LIN {X 0,Y 318.098,Z 206.968,A -85,B 0,C 180,E1 -15903.08,E2 -15903.08} C_VEL
LIN {X 0,Y 320.749,Z 222.526,A -85,B 0,C 180,E1 -15903.782,E2 -15903.782} C_VEL
LIN {X 0,Y 321.576,Z 229.62,A -85,B 0,C 180,E1 -15904.057,E2 -15904.057} C_VEL
LIN {X 0,Y 319.669,Z 290.634,A -85,B 0,C 180,E1 -15905.482,E2 -15905.482} C_VEL
LIN {X 0,Y 318.704,Z 303.737,A -85,B 0,C 180,E1 -15906.01,E2 -15906.01} C_VEL
LIN {X 0,Y 317.246,Z 316.408,A -85,B 0,C 180,E1 -15906.759,E2 -15906.759} C_VEL
LIN {X 0,Y 315.532,Z 328.526,A -85,B 0,C 180,E1 -15907.75,E2 -15907.75} C_VEL
LIN {X 0,Y 313.654,Z 340.033,A -85,B 0,C 180,E1 -15908.991,E2 -15908.991} C_VEL
LIN {X 0,Y 311.666,Z 350.433,A -85,B 0,C 180,E1 -15910.401,E2 -15910.401} C_VEL
LIN {X 0,Y 309.931,Z 358.976,A -85,B 0,C 180,E1 -15911.832,E2 -15911.832} C_VEL
LIN {X 0,Y 308.237,Z 367.598,A -85,B 0,C 180,E1 -15913.609,E2 -15913.609} C_VEL
LIN {X 0,Y 306.912,Z 374.656,A -85,B 0,C 180,E1 -15915.41,E2 -15915.41} C_VEL
LIN {X 0,Y 305.513,Z 380.916,A -85,B 0,C 180,E1 -15917.377,E2 -15917.377} C_VEL
LIN {X 0,Y 304.63,Z 385.925,A -85,B 0,C 180,E1 -15919.364,E2 -15919.364} C_VEL
LIN {X 0,Y 304.053,Z 389.825,A -85,B 0,C 180,E1 -15921.359,E2 -15921.359} C_VEL
LIN {X 0,Y 303.728,Z 392.717,A -85,B 0,C 180,E1 -15923.356,E2 -15923.356} C_VEL
LIN {X 0,Y 303.654,Z 395.096,A -85,B 0,C 180,E1 -15926.018,E2 -15926.018} C_VEL
LIN {X 0,Y 303.656,Z 395.702,A -85,B 0,C 180,E1 -15927.347,E2 -15927.347} C_VEL
LIN {X 0,Y 303.684,Z 395.883,A -85,B 0,C 180,E1 -15928.674,E2 -15928.674} C_VEL
LIN {X 0,Y 303.769,Z 395.655,A -85,B 0,C 180,E1 -15930,E2 -15930} C_VEL
LIN {X 0,Y 303.713,Z 395.029,A -85,B 0,C 180,E1 -15931.326,E2 -15931.326} C_VEL
LIN {X 0,Y 303.684,Z 394.007,A -85,B 0,C 180,E1 -15932.653,E2 -15932.653} C_VEL
LIN {X 0,Y 303.693,Z 392.539,A -85,B 0,C 180,E1 -15933.981,E2 -15933.981} C_VEL
LIN {X 0,Y 303.678,Z 390.075,A -85,B 0,C 180,E1 -15935.644,E2 -15935.644} C_VEL
LIN {X 0,Y 303.905,Z 385.397,A -85,B 0,C 180,E1 -15937.975,E2 -15937.975} C_VEL
LIN {X 0,Y 304.352,Z 379.061,A -85,B 0,C 180,E1 -15940.309,E2 -15940.309} C_VEL
LIN {X 0,Y 305.069,Z 372.151,A -85,B 0,C 180,E1 -15942.304,E2 -15942.304} C_VEL
LIN {X 0,Y 305.868,Z 365.084,A -85,B 0,C 180,E1 -15943.961,E2 -15943.961} C_VEL
LIN {X 0,Y 306.783,Z 357.329,A -85,B 0,C 180,E1 -15945.47,E2 -15945.47} C_VEL
LIN {X 0,Y 307.987,Z 347.315,A -85,B 0,C 180,E1 -15947.068,E2 -15947.068} C_VEL
LIN {X 0,Y 309.154,Z 336.997,A -85,B 0,C 180,E1 -15948.386,E2 -15948.386} C_VEL
LIN {X 0,Y 310.341,Z 325.889,A -85,B 0,C 180,E1 -15949.513,E2 -15949.513} C_VEL
LIN {X 0,Y 311.511,Z 313.595,A -85,B 0,C 180,E1 -15950.468,E2 -15950.468} C_VEL
LIN {X 0,Y 312.47,Z 300.68,A -85,B 0,C 180,E1 -15951.178,E2 -15951.178} C_VEL
LIN {X 0,Y 313.032,Z 286.986,A -85,B 0,C 180,E1 -15951.656,E2 -15951.656} C_VEL
LIN {X 0,Y 314.192,Z 225.236,A -85,B 0,C 180,E1 -15953.088,E2 -15953.088} C_VEL
LIN {X 0,Y 308.653,Z 182.969,A -85,B 0,C 180,E1 -15954.491,E2 -15954.491} C_VEL
LIN {X 0,Y 309.452,Z 175.908,A -85,B 0,C 180,E1 -15956.287,E2 -15956.287} C_VEL
LIN {X 0,Y 308.009,Z 167.396,A -85,B 0,C 180,E1 -15958.631,E2 -15958.631} C_VEL
LIN {X 0,Y 305.479,Z 155.435,A -85,B 0,C 180,E1 -15962.094,E2 -15962.094} C_VEL
LIN {X 0,Y 305.5,Z 155.431,A -85,B 0,C 180,E1 -15966.373,E2 -15966.373} C_VEL
LIN {X 0,Y 305.459,Z 155.436,A -85,B 0,C 180,E1 -15970.107,E2 -15970.107} C_VEL
LIN {X 0,Y 305.426,Z 155.442,A -85,B 0,C 180,E1 -15973.655,E2 -15973.655} C_VEL
LIN {X 0,Y 305.455,Z 155.437,A -85,B 0,C 180,E1 -15977.414,E2 -15977.414} C_VEL
LIN {X 0,Y 305.476,Z 155.437,A -85,B 0,C 180,E1 -15981.597,E2 -15981.597} C_VEL
LIN {X 0,Y 305.462,Z 155.434,A -85,B 0,C 180,E1 -15984.886,E2 -15984.886} C_VEL
LIN {X 0,Y 305.452,Z 155.434,A -85,B 0,C 180,E1 -15988.355,E2 -15988.355} C_VEL
LIN {X 0,Y 305.521,Z 155.429,A -85,B 0,C 180,E1 -15991.114,E2 -15991.114} C_VEL
LIN {X 0,Y 305.572,Z 155.419,A -85,B 0,C 180,E1 -15994.088,E2 -15994.088} C_VEL
LIN {X 0,Y 305.475,Z 155.429,A -85,B 0,C 180,E1 -15998.401,E2 -15998.401} C_VEL
LIN {X 0,Y 305.542,Z 155.417,A -85,B 0,C 180,E1 -16001.214,E2 -16001.214} C_VEL
LIN {X 0,Y 305.626,Z 155.412,A -85,B 0,C 180,E1 -16005.348,E2 -16005.348} C_VEL
LIN {X 0,Y 305.624,Z 155.413,A -85,B 0,C 180,E1 -16009.399,E2 -16009.399} C_VEL
LIN {X 0,Y 305.748,Z 155.396,A -85,B 0,C 180,E1 -16012.072,E2 -16012.072} C_VEL
LIN {X 0,Y 305.674,Z 155.407,A -85,B 0,C 180,E1 -16014.723,E2 -16014.723} C_VEL
LIN {X 0,Y 305.955,Z 155.375,A -85,B 0,C 180,E1 -16018.683,E2 -16018.683} C_VEL
LIN {X 0,Y 305.955,Z 155.368,A -85,B 0,C 180,E1 -16021.316,E2 -16021.316} C_VEL
LIN {X 0,Y 305.685,Z 155.404,A -85,B 0,C 180,E1 -16025.276,E2 -16025.276} C_VEL
LIN {X 0,Y 305.796,Z 155.391,A -85,B 0,C 180,E1 -16027.926,E2 -16027.926} C_VEL
LIN {X 0,Y 305.603,Z 155.412,A -85,B 0,C 180,E1 -16031.945,E2 -16031.945} C_VEL
LIN {X 0,Y 305.637,Z 155.411,A -85,B 0,C 180,E1 -16035.035,E2 -16035.035} C_VEL
LIN {X 0,Y 305.579,Z 155.418,A -85,B 0,C 180,E1 -16038.783,E2 -16038.783} C_VEL
LIN {X 0,Y 305.485,Z 155.428,A -85,B 0,C 180,E1 -16043.039,E2 -16043.039} C_VEL
LIN {X 0,Y 305.546,Z 155.426,A -85,B 0,C 180,E1 -16046.227,E2 -16046.227} C_VEL
LIN {X 0,Y 305.487,Z 155.427,A -85,B 0,C 180,E1 -16049.047,E2 -16049.047} C_VEL
LIN {X 0,Y 305.442,Z 155.438,A -85,B 0,C 180,E1 -16051.952,E2 -16051.952} C_VEL
LIN {X 0,Y 305.461,Z 155.432,A -85,B 0,C 180,E1 -16055.113,E2 -16055.113} C_VEL
LIN {X 0,Y 305.44,Z 155.433,A -85,B 0,C 180,E1 -16058.527,E2 -16058.527} C_VEL
LIN {X 0,Y 305.454,Z 155.433,A -85,B 0,C 180,E1 -16062.586,E2 -16062.586} C_VEL
LIN {X 0,Y 305.424,Z 155.437,A -85,B 0,C 180,E1 -16066.345,E2 -16066.345} C_VEL
LIN {X 0,Y 305.457,Z 155.435,A -85,B 0,C 180,E1 -16069.892,E2 -16069.892} C_VEL
LIN {X 0,Y 305.48,Z 155.434,A -85,B 0,C 180,E1 -16073.632,E2 -16073.632} C_VEL
LIN {X 0,Y 305.464,Z 155.431,A -85,B 0,C 180,E1 -16076.483,E2 -16076.483} C_VEL
LIN {X 0,Y 305.495,Z 155.43,A -85,B 0,C 180,E1 -16080.95,E2 -16080.95} C_VEL
LIN {X 0,Y 305.571,Z 155.418,A -85,B 0,C 180,E1 -16084.088,E2 -16084.088} C_VEL
LIN {X 0,Y 305.475,Z 155.432,A -85,B 0,C 180,E1 -16088.401,E2 -16088.401} C_VEL
LIN {X 0,Y 305.542,Z 155.425,A -85,B 0,C 180,E1 -16091.215,E2 -16091.215} C_VEL
LIN {X 0,Y 305.626,Z 155.414,A -85,B 0,C 180,E1 -16095.348,E2 -16095.348} C_VEL
LIN {X 0,Y 305.624,Z 155.414,A -85,B 0,C 180,E1 -16099.399,E2 -16099.399} C_VEL
LIN {X 0,Y 305.748,Z 155.395,A -85,B 0,C 180,E1 -16102.073,E2 -16102.073} C_VEL
LIN {X 0,Y 305.674,Z 155.541,A -85,B 0,C 180,E1 -16104.889,E2 -16104.889} C_VEL
LIN {X 0,Y 306.008,Z 157.231,A -85,B 0,C 180,E1 -16105.424,E2 -16105.424} C_VEL
LIN {X 0,Y 313.1,Z 177.176,A -85,B 0,C 180,E1 -16106.405,E2 -16106.405} C_VEL
LIN {X 0,Y 314.55,Z 182.856,A -85,B 0,C 180,E1 -16106.637,E2 -16106.637} C_VEL
LIN {X 0,Y 315.065,Z 186.672,A -85,B 0,C 180,E1 -16106.763,E2 -16106.763} C_VEL
LIN {X 0,Y 313.152,Z 265.366,A -85,B 0,C 180,E1 -16108.599,E2 -16108.599} C_VEL
LIN {X 0,Y 312.585,Z 278.914,A -85,B 0,C 180,E1 -16109.195,E2 -16109.195} C_VEL
LIN {X 0,Y 311.853,Z 291.275,A -85,B 0,C 180,E1 -16110,E2 -16110} C_VEL
LIN {X 0,Y 310.932,Z 302.407,A -85,B 0,C 180,E1 -16110.972,E2 -16110.972} C_VEL
LIN {X 0,Y 309.759,Z 313.993,A -85,B 0,C 180,E1 -16112.269,E2 -16112.269} C_VEL
LIN {X 0,Y 308.583,Z 324.524,A -85,B 0,C 180,E1 -16113.755,E2 -16113.755} C_VEL
LIN {X 0,Y 307.513,Z 333.085,A -85,B 0,C 180,E1 -16115.245,E2 -16115.245} C_VEL
LIN {X 0,Y 306.334,Z 342.342,A -85,B 0,C 180,E1 -16117.249,E2 -16117.249} C_VEL
LIN {X 0,Y 305.428,Z 349.79,A -85,B 0,C 180,E1 -16119.269,E2 -16119.269} C_VEL
LIN {X 0,Y 304.727,Z 355.732,A -85,B 0,C 180,E1 -16121.306,E2 -16121.306} C_VEL
LIN {X 0,Y 304.265,Z 360.38,A -85,B 0,C 180,E1 -16123.355,E2 -16123.355} C_VEL
LIN {X 0,Y 303.862,Z 363.912,A -85,B 0,C 180,E1 -16125.426,E2 -16125.426} C_VEL
LIN {X 0,Y 303.599,Z 367.109,A -85,B 0,C 180,E1 -16128.359,E2 -16128.359} C_VEL
LIN {X 0,Y 303.554,Z 368.119,A -85,B 0,C 180,E1 -16130.322,E2 -16130.322} C_VEL
LIN {X 0,Y 303.691,Z 368.27,A -85,B 0,C 180,E1 -16132.23,E2 -16132.23} C_VEL
LIN {X 0,Y 304.02,Z 367.364,A -85,B 0,C 180,E1 -16134.589,E2 -16134.589} C_VEL
LIN {X 0,Y 304.337,Z 366.189,A -85,B 0,C 180,E1 -16136.025,E2 -16136.025} C_VEL
LIN {X 0,Y 305.026,Z 363.501,A -85,B 0,C 180,E1 -16138.186,E2 -16138.186} C_VEL
LIN {X 0,Y 305.938,Z 359.612,A -85,B 0,C 180,E1 -16140.357,E2 -16140.357} C_VEL
LIN {X 0,Y 307.175,Z 354.217,A -85,B 0,C 180,E1 -16142.593,E2 -16142.593} C_VEL
LIN {X 0,Y 308.695,Z 347.638,A -85,B 0,C 180,E1 -16144.693,E2 -16144.693} C_VEL
LIN {X 0,Y 310.26,Z 340.559,A -85,B 0,C 180,E1 -16146.485,E2 -16146.485} C_VEL
LIN {X 0,Y 312.107,Z 331.396,A -85,B 0,C 180,E1 -16148.354,E2 -16148.354} C_VEL
LIN {X 0,Y 313.882,Z 322.187,A -85,B 0,C 180,E1 -16149.861,E2 -16149.861} C_VEL
LIN {X 0,Y 315.728,Z 311.658,A -85,B 0,C 180,E1 -16151.245,E2 -16151.245} C_VEL
LIN {X 0,Y 317.434,Z 299.665,A -85,B 0,C 180,E1 -16152.476,E2 -16152.476} C_VEL
LIN {X 0,Y 318.779,Z 287.425,A -85,B 0,C 180,E1 -16153.438,E2 -16153.438} C_VEL
LIN {X 0,Y 319.871,Z 274.616,A -85,B 0,C 180,E1 -16154.151,E2 -16154.151} C_VEL
LIN {X 0,Y 320.505,Z 261.159,A -85,B 0,C 180,E1 -16154.635,E2 -16154.635} C_VEL
LIN {X 0,Y 322.56,Z 192.231,A -85,B 0,C 180,E1 -16156.232,E2 -16156.232} C_VEL
LIN {X 0,Y 316.448,Z 178.489,A -85,B 0,C 180,E1 -16157.287,E2 -16157.287} C_VEL
LIN {X 0,Y 316.128,Z 177.812,A -85,B 0,C 180,E1 -16157.343,E2 -16157.343} C_VEL
LIN {X 0,Y 314.073,Z 174.928,A -85,B 0,C 180,E1 -16157.664,E2 -16157.664} C_VEL
LIN {X 0,Y 309.469,Z 171.568,A -85,B 0,C 180,E1 -16158.319,E2 -16158.319} C_VEL
LIN {X 0,Y 304.78,Z 168.323,A -85,B 0,C 180,E1 -16159.01,E2 -16159.01} C_VEL
LIN {X 0,Y 302.586,Z 165.592,A -85,B 0,C 180,E1 -16159.38,E2 -16159.38} C_VEL
LIN {X 0,Y 299.095,Z 159.067,A -85,B 0,C 180,E1 -16160.076,E2 -16160.076} C_VEL
LIN {X 0,Y 298.387,Z 156.315,A -85,B 0,C 180,E1 -16161.212,E2 -16161.212} C_VEL
LIN {X 0,Y 298.404,Z 156.303,A -85,B 0,C 180,E1 -16163.928,E2 -16163.928} C_VEL
LIN {X 0,Y 298.393,Z 156.318,A -85,B 0,C 180,E1 -16167.2,E2 -16167.2} C_VEL
LIN {X 0,Y 298.365,Z 156.321,A -85,B 0,C 180,E1 -16170.638,E2 -16170.638} C_VEL
LIN {X 0,Y 298.413,Z 156.312,A -85,B 0,C 180,E1 -16174.918,E2 -16174.918} C_VEL
LIN {X 0,Y 298.389,Z 156.309,A -85,B 0,C 180,E1 -16177.862,E2 -16177.862} C_VEL
LIN {X 0,Y 298.451,Z 156.301,A -85,B 0,C 180,E1 -16180.751,E2 -16180.751} C_VEL
LIN {X 0,Y 298.511,Z 156.292,A -85,B 0,C 180,E1 -16184.991,E2 -16184.991} C_VEL
LIN {X 0,Y 298.578,Z 156.28,A -85,B 0,C 180,E1 -16189.146,E2 -16189.146} C_VEL
LIN {X 0,Y 298.7,Z 156.276,A -85,B 0,C 180,E1 -16191.885,E2 -16191.885} C_VEL
LIN {X 0,Y 298.626,Z 156.28,A -85,B 0,C 180,E1 -16194.599,E2 -16194.599} C_VEL
LIN {X 0,Y 298.903,Z 156.24,A -85,B 0,C 180,E1 -16198.653,E2 -16198.653} C_VEL
LIN {X 0,Y 298.904,Z 156.25,A -85,B 0,C 180,E1 -16201.348,E2 -16201.348} C_VEL
LIN {X 0,Y 298.736,Z 156.268,A -85,B 0,C 180,E1 -16206.756,E2 -16206.756} C_VEL
LIN {X 0,Y 298.627,Z 156.283,A -85,B 0,C 180,E1 -16209.482,E2 -16209.482} C_VEL
LIN {X 0,Y 298.547,Z 156.286,A -85,B 0,C 180,E1 -16213.616,E2 -16213.616} C_VEL
LIN {X 0,Y 298.489,Z 156.3,A -85,B 0,C 180,E1 -16216.412,E2 -16216.412} C_VEL
LIN {X 0,Y 298.489,Z 156.304,A -85,B 0,C 180,E1 -16219.641,E2 -16219.641} C_VEL
LIN {X 0,Y 298.425,Z 156.308,A -85,B 0,C 180,E1 -16223.601,E2 -16223.601} C_VEL
LIN {X 0,Y 298.41,Z 156.303,A -85,B 0,C 180,E1 -16226.582,E2 -16226.582} C_VEL
LIN {X 0,Y 298.396,Z 156.31,A -85,B 0,C 180,E1 -16229.644,E2 -16229.644} C_VEL
LIN {X 0,Y 298.395,Z 156.316,A -85,B 0,C 180,E1 -16232.801,E2 -16232.801} C_VEL
LIN {X 0,Y 298.43,Z 156.307,A -85,B 0,C 180,E1 -16236.803,E2 -16236.803} C_VEL
LIN {X 0,Y 298.376,Z 156.318,A -85,B 0,C 180,E1 -16239.492,E2 -16239.492} C_VEL
LIN {X 0,Y 298.373,Z 156.317,A -85,B 0,C 180,E1 -16243.098,E2 -16243.098} C_VEL
LIN {X 0,Y 298.405,Z 156.32,A -85,B 0,C 180,E1 -16246.921,E2 -16246.921} C_VEL
LIN {X 0,Y 298.406,Z 156.317,A -85,B 0,C 180,E1 -16251.006,E2 -16251.006} C_VEL
LIN {X 0,Y 298.454,Z 156.374,A -85,B 0,C 180,E1 -16252.141,E2 -16252.141} C_VEL
LIN {X 0,Y 301.266,Z 166.786,A -85,B 0,C 180,E1 -16255.952,E2 -16255.952} C_VEL
LIN {X 0,Y 303.943,Z 178.256,A -85,B 0,C 180,E1 -16259.807,E2 -16259.807} C_VEL
LIN {X 0,Y 304.513,Z 181.202,A -85,B 0,C 180,E1 -16260.744,E2 -16260.744} C_VEL
LIN {X 0,Y 308.356,Z 190.471,A -85,B 0,C 180,E1 -16261.494,E2 -16261.494} C_VEL
LIN {X 0,Y 311.822,Z 206.926,A -85,B 0,C 180,E1 -16262.365,E2 -16262.365} C_VEL
LIN {X 0,Y 314.608,Z 223.163,A -85,B 0,C 180,E1 -16263.126,E2 -16263.126} C_VEL
LIN {X 0,Y 315.47,Z 230.001,A -85,B 0,C 180,E1 -16263.407,E2 -16263.407} C_VEL
LIN {X 0,Y 313.534,Z 290.112,A -85,B 0,C 180,E1 -16264.837,E2 -16264.837} C_VEL
LIN {X 0,Y 312.525,Z 303.285,A -85,B 0,C 180,E1 -16265.372,E2 -16265.372} C_VEL
LIN {X 0,Y 311.087,Z 315.427,A -85,B 0,C 180,E1 -16266.094,E2 -16266.094} C_VEL
LIN {X 0,Y 309.534,Z 326.016,A -85,B 0,C 180,E1 -16266.942,E2 -16266.942} C_VEL
LIN {X 0,Y 308.04,Z 335.282,A -85,B 0,C 180,E1 -16267.886,E2 -16267.886} C_VEL
LIN {X 0,Y 305.94,Z 346.581,A -85,B 0,C 180,E1 -16269.317,E2 -16269.317} C_VEL
LIN {X 0,Y 303.98,Z 355.709,A -85,B 0,C 180,E1 -16270.764,E2 -16270.764} C_VEL
LIN {X 0,Y 301.99,Z 364.922,A -85,B 0,C 180,E1 -16272.587,E2 -16272.587} C_VEL
LIN {X 0,Y 300.528,Z 372.301,A -85,B 0,C 180,E1 -16274.399,E2 -16274.399} C_VEL
LIN {X 0,Y 299.005,Z 378.958,A -85,B 0,C 180,E1 -16276.405,E2 -16276.405} C_VEL
LIN {X 0,Y 297.881,Z 384.307,A -85,B 0,C 180,E1 -16278.431,E2 -16278.431} C_VEL
LIN {X 0,Y 297.197,Z 388.504,A -85,B 0,C 180,E1 -16280.472,E2 -16280.472} C_VEL
LIN {X 0,Y 296.867,Z 390.741,A -85,B 0,C 180,E1 -16281.834,E2 -16281.834} C_VEL
LIN {X 0,Y 296.553,Z 393.862,A -85,B 0,C 180,E1 -16284.56,E2 -16284.56} C_VEL
LIN {X 0,Y 296.568,Z 394.833,A -85,B 0,C 180,E1 -16285.923,E2 -16285.923} C_VEL
LIN {X 0,Y 296.579,Z 395.406,A -85,B 0,C 180,E1 -16287.283,E2 -16287.283} C_VEL
LIN {X 0,Y 296.597,Z 395.544,A -85,B 0,C 180,E1 -16288.642,E2 -16288.642} C_VEL
LIN {X 0,Y 296.677,Z 395.291,A -85,B 0,C 180,E1 -16290,E2 -16290} C_VEL
LIN {X 0,Y 296.625,Z 394.64,A -85,B 0,C 180,E1 -16291.357,E2 -16291.357} C_VEL
LIN {X 0,Y 296.607,Z 393.588,A -85,B 0,C 180,E1 -16292.716,E2 -16292.716} C_VEL
LIN {X 0,Y 296.606,Z 392.071,A -85,B 0,C 180,E1 -16294.076,E2 -16294.076} C_VEL
LIN {X 0,Y 296.613,Z 388.985,A -85,B 0,C 180,E1 -16296.12,E2 -16296.12} C_VEL
LIN {X 0,Y 296.843,Z 384.814,A -85,B 0,C 180,E1 -16298.167,E2 -16298.167} C_VEL
LIN {X 0,Y 297.33,Z 378.412,A -85,B 0,C 180,E1 -16300.555,E2 -16300.555} C_VEL
LIN {X 0,Y 298.114,Z 371.432,A -85,B 0,C 180,E1 -16302.595,E2 -16302.595} C_VEL
LIN {X 0,Y 299.16,Z 362.658,A -85,B 0,C 180,E1 -16304.628,E2 -16304.628} C_VEL
LIN {X 0,Y 300.164,Z 353.634,A -85,B 0,C 180,E1 -16306.318,E2 -16306.318} C_VEL
LIN {X 0,Y 301.441,Z 343.735,A -85,B 0,C 180,E1 -16307.818,E2 -16307.818} C_VEL
LIN {X 0,Y 302.705,Z 332.818,A -85,B 0,C 180,E1 -16309.144,E2 -16309.144} C_VEL
LIN {X 0,Y 303.992,Z 320.561,A -85,B 0,C 180,E1 -16310.291,E2 -16310.291} C_VEL
LIN {X 0,Y 305.12,Z 307.747,A -85,B 0,C 180,E1 -16311.182,E2 -16311.182} C_VEL
LIN {X 0,Y 305.952,Z 294.977,A -85,B 0,C 180,E1 -16311.785,E2 -16311.785} C_VEL
LIN {X 0,Y 306.484,Z 277.039,A -85,B 0,C 180,E1 -16312.276,E2 -16312.276} C_VEL
LIN {X 0,Y 307.417,Z 225.576,A -85,B 0,C 180,E1 -16313.496,E2 -16313.496} C_VEL
LIN {X 0,Y 301.792,Z 182.64,A -85,B 0,C 180,E1 -16314.964,E2 -16314.964} C_VEL
LIN {X 0,Y 302.448,Z 176.485,A -85,B 0,C 180,E1 -16316.571,E2 -16316.571} C_VEL
LIN {X 0,Y 300.628,Z 166.507,A -85,B 0,C 180,E1 -16319.402,E2 -16319.402} C_VEL
LIN {X 0,Y 298.437,Z 156.311,A -85,B 0,C 180,E1 -16322.464,E2 -16322.464} C_VEL
LIN {X 0,Y 298.452,Z 156.308,A -85,B 0,C 180,E1 -16326.808,E2 -16326.808} C_VEL
LIN {X 0,Y 298.41,Z 156.314,A -85,B 0,C 180,E1 -16329.486,E2 -16329.486} C_VEL
LIN {X 0,Y 298.399,Z 156.313,A -85,B 0,C 180,E1 -16333.103,E2 -16333.103} C_VEL
LIN {X 0,Y 298.403,Z 156.313,A -85,B 0,C 180,E1 -16336.92,E2 -16336.92} C_VEL
LIN {X 0,Y 298.405,Z 156.314,A -85,B 0,C 180,E1 -16341.006,E2 -16341.006} C_VEL
LIN {X 0,Y 298.419,Z 156.312,A -85,B 0,C 180,E1 -16343.93,E2 -16343.93} C_VEL
LIN {X 0,Y 298.395,Z 156.314,A -85,B 0,C 180,E1 -16347.983,E2 -16347.983} C_VEL
LIN {X 0,Y 298.47,Z 156.305,A -85,B 0,C 180,E1 -16351.905,E2 -16351.905} C_VEL
LIN {X 0,Y 298.485,Z 156.304,A -85,B 0,C 180,E1 -16354.924,E2 -16354.924} C_VEL
LIN {X 0,Y 298.429,Z 156.306,A -85,B 0,C 180,E1 -16359.313,E2 -16359.313} C_VEL
LIN {X 0,Y 298.477,Z 156.291,A -85,B 0,C 180,E1 -16362.175,E2 -16362.175} C_VEL
LIN {X 0,Y 298.585,Z 156.287,A -85,B 0,C 180,E1 -16364.994,E2 -16364.994} C_VEL
LIN {X 0,Y 298.583,Z 156.292,A -85,B 0,C 180,E1 -16369.146,E2 -16369.146} C_VEL
LIN {X 0,Y 298.699,Z 156.273,A -85,B 0,C 180,E1 -16371.884,E2 -16371.884} C_VEL
LIN {X 0,Y 298.642,Z 156.281,A -85,B 0,C 180,E1 -16374.598,E2 -16374.598} C_VEL
LIN {X 0,Y 298.922,Z 156.251,A -85,B 0,C 180,E1 -16378.653,E2 -16378.653} C_VEL
LIN {X 0,Y 298.922,Z 156.244,A -85,B 0,C 180,E1 -16381.347,E2 -16381.347} C_VEL
LIN {X 0,Y 298.787,Z 156.267,A -85,B 0,C 180,E1 -16386.754,E2 -16386.754} C_VEL
LIN {X 0,Y 298.635,Z 156.281,A -85,B 0,C 180,E1 -16389.482,E2 -16389.482} C_VEL
LIN {X 0,Y 298.551,Z 156.292,A -85,B 0,C 180,E1 -16393.615,E2 -16393.615} C_VEL
LIN {X 0,Y 298.548,Z 156.298,A -85,B 0,C 180,E1 -16396.408,E2 -16396.408} C_VEL
LIN {X 0,Y 298.497,Z 156.299,A -85,B 0,C 180,E1 -16399.647,E2 -16399.647} C_VEL
LIN {X 0,Y 298.427,Z 156.308,A -85,B 0,C 180,E1 -16403.6,E2 -16403.6} C_VEL
LIN {X 0,Y 298.488,Z 156.302,A -85,B 0,C 180,E1 -16406.574,E2 -16406.574} C_VEL
LIN {X 0,Y 298.415,Z 156.31,A -85,B 0,C 180,E1 -16409.641,E2 -16409.641} C_VEL
LIN {X 0,Y 298.394,Z 156.312,A -85,B 0,C 180,E1 -16412.8,E2 -16412.8} C_VEL
LIN {X 0,Y 298.443,Z 156.305,A -85,B 0,C 180,E1 -16416.807,E2 -16416.807} C_VEL
LIN {X 0,Y 298.386,Z 156.314,A -85,B 0,C 180,E1 -16421.088,E2 -16421.088} C_VEL
LIN {X 0,Y 298.397,Z 156.313,A -85,B 0,C 180,E1 -16423.103,E2 -16423.103} C_VEL
LIN {X 0,Y 298.401,Z 156.311,A -85,B 0,C 180,E1 -16426.921,E2 -16426.921} C_VEL
LIN {X 0,Y 298.403,Z 156.312,A -85,B 0,C 180,E1 -16431.006,E2 -16431.006} C_VEL
LIN {X 0,Y 298.417,Z 156.312,A -85,B 0,C 180,E1 -16433.93,E2 -16433.93} C_VEL
LIN {X 0,Y 298.394,Z 156.309,A -85,B 0,C 180,E1 -16437.984,E2 -16437.984} C_VEL
LIN {X 0,Y 298.469,Z 156.305,A -85,B 0,C 180,E1 -16441.905,E2 -16441.905} C_VEL
LIN {X 0,Y 298.484,Z 156.304,A -85,B 0,C 180,E1 -16444.924,E2 -16444.924} C_VEL
LIN {X 0,Y 298.428,Z 156.312,A -85,B 0,C 180,E1 -16449.314,E2 -16449.314} C_VEL
LIN {X 0,Y 298.503,Z 156.299,A -85,B 0,C 180,E1 -16452.177,E2 -16452.177} C_VEL
LIN {X 0,Y 298.585,Z 156.293,A -85,B 0,C 180,E1 -16454.995,E2 -16454.995} C_VEL
LIN {X 0,Y 298.583,Z 156.293,A -85,B 0,C 180,E1 -16459.146,E2 -16459.146} C_VEL
LIN {X 0,Y 298.699,Z 156.273,A -85,B 0,C 180,E1 -16461.885,E2 -16461.885} C_VEL
LIN {X 0,Y 298.673,Z 156.406,A -85,B 0,C 180,E1 -16464.557,E2 -16464.557} C_VEL
LIN {X 0,Y 298.922,Z 157.762,A -85,B 0,C 180,E1 -16464.952,E2 -16464.952} C_VEL
LIN {X 0,Y 306.712,Z 179.512,A -85,B 0,C 180,E1 -16466.04,E2 -16466.04} C_VEL
LIN {X 0,Y 307.949,Z 184.293,A -85,B 0,C 180,E1 -16466.243,E2 -16466.243} C_VEL
LIN {X 0,Y 308.347,Z 188.503,A -85,B 0,C 180,E1 -16466.374,E2 -16466.374} C_VEL
LIN {X 0,Y 306.41,Z 265.138,A -85,B 0,C 180,E1 -16468.193,E2 -16468.193} C_VEL
LIN {X 0,Y 305.813,Z 278.957,A -85,B 0,C 180,E1 -16468.807,E2 -16468.807} C_VEL
LIN {X 0,Y 305.031,Z 291.905,A -85,B 0,C 180,E1 -16469.67,E2 -16469.67} C_VEL
LIN {X 0,Y 303.899,Z 304.584,A -85,B 0,C 180,E1 -16470.828,E2 -16470.828} C_VEL
LIN {X 0,Y 302.711,Z 316.164,A -85,B 0,C 180,E1 -16472.202,E2 -16472.202} C_VEL
LIN {X 0,Y 301.514,Z 326.011,A -85,B 0,C 180,E1 -16473.675,E2 -16473.675} C_VEL
LIN {X 0,Y 300.282,Z 335.212,A -85,B 0,C 180,E1 -16475.372,E2 -16475.372} C_VEL
LIN {X 0,Y 299.149,Z 344.155,A -85,B 0,C 180,E1 -16477.424,E2 -16477.424} C_VEL
LIN {X 0,Y 298.276,Z 351.264,A -85,B 0,C 180,E1 -16479.494,E2 -16479.494} C_VEL
LIN {X 0,Y 297.557,Z 356.959,A -85,B 0,C 180,E1 -16481.582,E2 -16481.582} C_VEL
LIN {X 0,Y 297.032,Z 362.083,A -85,B 0,C 180,E1 -16484.05,E2 -16484.05} C_VEL
LIN {X 0,Y 296.598,Z 365.638,A -85,B 0,C 180,E1 -16486.52,E2 -16486.52} C_VEL
LIN {X 0,Y 296.5,Z 367.509,A -85,B 0,C 180,E1 -16488.536,E2 -16488.536} C_VEL
LIN {X 0,Y 296.478,Z 368.542,A -85,B 0,C 180,E1 -16490.829,E2 -16490.829} C_VEL
LIN {X 0,Y 296.628,Z 368.591,A -85,B 0,C 180,E1 -16492.478,E2 -16492.478} C_VEL
LIN {X 0,Y 296.764,Z 368.255,A -85,B 0,C 180,E1 -16493.741,E2 -16493.741} C_VEL
LIN {X 0,Y 297.258,Z 366.743,A -85,B 0,C 180,E1 -16496.049,E2 -16496.049} C_VEL
LIN {X 0,Y 297.918,Z 364.327,A -85,B 0,C 180,E1 -16498.152,E2 -16498.152} C_VEL
LIN {X 0,Y 298.871,Z 360.641,A -85,B 0,C 180,E1 -16500.37,E2 -16500.37} C_VEL
LIN {X 0,Y 300.079,Z 355.62,A -85,B 0,C 180,E1 -16502.594,E2 -16502.594} C_VEL
LIN {X 0,Y 301.689,Z 349.113,A -85,B 0,C 180,E1 -16504.802,E2 -16504.802} C_VEL
LIN {X 0,Y 303.273,Z 342.322,A -85,B 0,C 180,E1 -16506.636,E2 -16506.636} C_VEL
LIN {X 0,Y 305.132,Z 334.002,A -85,B 0,C 180,E1 -16508.454,E2 -16508.454} C_VEL
LIN {X 0,Y 307.016,Z 324.737,A -85,B 0,C 180,E1 -16510.077,E2 -16510.077} C_VEL
LIN {X 0,Y 308.939,Z 314.623,A -85,B 0,C 180,E1 -16511.496,E2 -16511.496} C_VEL
LIN {X 0,Y 310.692,Z 303.571,A -85,B 0,C 180,E1 -16512.736,E2 -16512.736} C_VEL
LIN {X 0,Y 312.082,Z 292.113,A -85,B 0,C 180,E1 -16513.746,E2 -16513.746} C_VEL
LIN {X 0,Y 313.307,Z 279.378,A -85,B 0,C 180,E1 -16514.563,E2 -16514.563} C_VEL
LIN {X 0,Y 314.171,Z 266.021,A -85,B 0,C 180,E1 -16515.142,E2 -16515.142} C_VEL
LIN {X 0,Y 316.545,Z 194.382,A -85,B 0,C 180,E1 -16516.845,E2 -16516.845} C_VEL
LIN {X 0,Y 310.69,Z 181.273,A -85,B 0,C 180,E1 -16517.892,E2 -16517.892} C_VEL
LIN {X 0,Y 303.113,Z 166.457,A -85,B 0,C 180,E1 -16519.284,E2 -16519.284} C_VEL
LIN {X 0,Y 302.586,Z 165.592,A -85,B 0,C 180,E1 -16519.38,E2 -16519.38} C_VEL
LIN {X 0,Y 300.332,Z 162.641,A -85,B 0,C 180,E1 -16519.773,E2 -16519.773} C_VEL
LIN {X 0,Y 297.61,Z 160.433,A -85,B 0,C 180,E1 -16520.245,E2 -16520.245} C_VEL
LIN {X 0,Y 294.935,Z 158.937,A -85,B 0,C 180,E1 -16520.802,E2 -16520.802} C_VEL
LIN {X 0,Y 292.154,Z 157.819,A -85,B 0,C 180,E1 -16521.698,E2 -16521.698} C_VEL
LIN {X 0,Y 291.36,Z 157.194,A -85,B 0,C 180,E1 -16522.407,E2 -16522.407} C_VEL
LIN {X 0,Y 291.357,Z 157.186,A -85,B 0,C 180,E1 -16522.474,E2 -16522.474} C_VEL
LIN {X 0,Y 291.344,Z 157.193,A -85,B 0,C 180,E1 -16526.302,E2 -16526.302} C_VEL
LIN {X 0,Y 291.335,Z 157.2,A -85,B 0,C 180,E1 -16530.279,E2 -16530.279} C_VEL
LIN {X 0,Y 291.342,Z 157.192,A -85,B 0,C 180,E1 -16534.265,E2 -16534.265} C_VEL
LIN {X 0,Y 291.349,Z 157.187,A -85,B 0,C 180,E1 -16537.297,E2 -16537.297} C_VEL
LIN {X 0,Y 291.385,Z 157.185,A -85,B 0,C 180,E1 -16540.265,E2 -16540.265} C_VEL
LIN {X 0,Y 291.452,Z 157.171,A -85,B 0,C 180,E1 -16544.699,E2 -16544.699} C_VEL
LIN {X 0,Y 291.522,Z 157.16,A -85,B 0,C 180,E1 -16548.88,E2 -16548.88} C_VEL
LIN {X 0,Y 291.653,Z 157.156,A -85,B 0,C 180,E1 -16551.687,E2 -16551.687} C_VEL
LIN {X 0,Y 291.596,Z 157.154,A -85,B 0,C 180,E1 -16554.468,E2 -16554.468} C_VEL
LIN {X 0,Y 291.87,Z 157.116,A -85,B 0,C 180,E1 -16558.621,E2 -16558.621} C_VEL
LIN {X 0,Y 291.871,Z 157.125,A -85,B 0,C 180,E1 -16561.38,E2 -16561.38} C_VEL
LIN {X 0,Y 291.688,Z 157.143,A -85,B 0,C 180,E1 -16566.92,E2 -16566.92} C_VEL
LIN {X 0,Y 291.57,Z 157.164,A -85,B 0,C 180,E1 -16569.714,E2 -16569.714} C_VEL
LIN {X 0,Y 291.517,Z 157.165,A -85,B 0,C 180,E1 -16573.951,E2 -16573.951} C_VEL
LIN {X 0,Y 291.444,Z 157.17,A -85,B 0,C 180,E1 -16578.27,E2 -16578.27} C_VEL
LIN {X 0,Y 291.364,Z 157.183,A -85,B 0,C 180,E1 -16581.212,E2 -16581.212} C_VEL
LIN {X 0,Y 291.366,Z 157.189,A -85,B 0,C 180,E1 -16584.209,E2 -16584.209} C_VEL
LIN {X 0,Y 291.356,Z 157.184,A -85,B 0,C 180,E1 -16587.279,E2 -16587.279} C_VEL
LIN {X 0,Y 291.32,Z 157.188,A -85,B 0,C 180,E1 -16590.439,E2 -16590.439} C_VEL
LIN {X 0,Y 291.346,Z 157.187,A -85,B 0,C 180,E1 -16593.699,E2 -16593.699} C_VEL
LIN {X 0,Y 291.361,Z 157.186,A -85,B 0,C 180,E1 -16597.25,E2 -16597.25} C_VEL
LIN {X 0,Y 291.302,Z 157.196,A -85,B 0,C 180,E1 -16600.648,E2 -16600.648} C_VEL
LIN {X 0,Y 291.284,Z 157.206,A -85,B 0,C 180,E1 -16604.404,E2 -16604.404} C_VEL
LIN {X 0,Y 291.329,Z 157.198,A -85,B 0,C 180,E1 -16608.404,E2 -16608.404} C_VEL
LIN {X 0,Y 291.397,Z 157.312,A -85,B 0,C 180,E1 -16611.269,E2 -16611.269} C_VEL
LIN {X 0,Y 294.085,Z 167.027,A -85,B 0,C 180,E1 -16615.002,E2 -16615.002} C_VEL
LIN {X 0,Y 296.198,Z 175.934,A -85,B 0,C 180,E1 -16618.134,E2 -16618.134} C_VEL
LIN {X 0,Y 297.297,Z 180.786,A -85,B 0,C 180,E1 -16619.765,E2 -16619.765} C_VEL
LIN {X 0,Y 302.53,Z 192.539,A -85,B 0,C 180,E1 -16620.815,E2 -16620.815} C_VEL
LIN {X 0,Y 305.491,Z 206.319,A -85,B 0,C 180,E1 -16621.591,E2 -16621.591} C_VEL
LIN {X 0,Y 308.697,Z 225.105,A -85,B 0,C 180,E1 -16622.502,E2 -16622.502} C_VEL
LIN {X 0,Y 309.371,Z 231.526,A -85,B 0,C 180,E1 -16622.759,E2 -16622.759} C_VEL
LIN {X 0,Y 307.424,Z 289.568,A -85,B 0,C 180,E1 -16624.163,E2 -16624.163} C_VEL
LIN {X 0,Y 306.38,Z 302.835,A -85,B 0,C 180,E1 -16624.707,E2 -16624.707} C_VEL
LIN {X 0,Y 304.813,Z 315.565,A -85,B 0,C 180,E1 -16625.479,E2 -16625.479} C_VEL
LIN {X 0,Y 303.071,Z 326.924,A -85,B 0,C 180,E1 -16626.421,E2 -16626.421} C_VEL
LIN {X 0,Y 301.325,Z 337.335,A -85,B 0,C 180,E1 -16627.547,E2 -16627.547} C_VEL
LIN {X 0,Y 299.082,Z 348.088,A -85,B 0,C 180,E1 -16629.001,E2 -16629.001} C_VEL
LIN {X 0,Y 296.892,Z 357.788,A -85,B 0,C 180,E1 -16630.646,E2 -16630.646} C_VEL
LIN {X 0,Y 295.137,Z 365.546,A -85,B 0,C 180,E1 -16632.272,E2 -16632.272} C_VEL
LIN {X 0,Y 293.439,Z 373.63,A -85,B 0,C 180,E1 -16634.369,E2 -16634.369} C_VEL
LIN {X 0,Y 291.627,Z 380.862,A -85,B 0,C 180,E1 -16636.765,E2 -16636.765} C_VEL
LIN {X 0,Y 290.625,Z 385.734,A -85,B 0,C 180,E1 -16638.845,E2 -16638.845} C_VEL
LIN {X 0,Y 289.983,Z 389.51,A -85,B 0,C 180,E1 -16640.936,E2 -16640.936} C_VEL
LIN {X 0,Y 289.578,Z 392.29,A -85,B 0,C 180,E1 -16643.03,E2 -16643.03} C_VEL
LIN {X 0,Y 289.466,Z 394.568,A -85,B 0,C 180,E1 -16645.823,E2 -16645.823} C_VEL
LIN {X 0,Y 289.504,Z 395.097,A -85,B 0,C 180,E1 -16647.217,E2 -16647.217} C_VEL
LIN {X 0,Y 289.513,Z 395.206,A -85,B 0,C 180,E1 -16648.609,E2 -16648.609} C_VEL
LIN {X 0,Y 289.587,Z 394.928,A -85,B 0,C 180,E1 -16650,E2 -16650} C_VEL
LIN {X 0,Y 289.539,Z 394.252,A -85,B 0,C 180,E1 -16651.391,E2 -16651.391} C_VEL
LIN {X 0,Y 289.531,Z 393.157,A -85,B 0,C 180,E1 -16652.782,E2 -16652.782} C_VEL
LIN {X 0,Y 289.522,Z 391.604,A -85,B 0,C 180,E1 -16654.176,E2 -16654.176} C_VEL
LIN {X 0,Y 289.548,Z 388.461,A -85,B 0,C 180,E1 -16656.27,E2 -16656.27} C_VEL
LIN {X 0,Y 289.774,Z 384.229,A -85,B 0,C 180,E1 -16658.367,E2 -16658.367} C_VEL
LIN {X 0,Y 290.306,Z 377.763,A -85,B 0,C 180,E1 -16660.814,E2 -16660.814} C_VEL
LIN {X 0,Y 291.164,Z 370.696,A -85,B 0,C 180,E1 -16662.901,E2 -16662.901} C_VEL
LIN {X 0,Y 292.269,Z 361.811,A -85,B 0,C 180,E1 -16664.981,E2 -16664.981} C_VEL
LIN {X 0,Y 293.316,Z 352.681,A -85,B 0,C 180,E1 -16666.71,E2 -16666.71} C_VEL
LIN {X 0,Y 294.586,Z 342.636,A -85,B 0,C 180,E1 -16668.247,E2 -16668.247} C_VEL
LIN {X 0,Y 295.885,Z 331.458,A -85,B 0,C 180,E1 -16669.603,E2 -16669.603} C_VEL
LIN {X 0,Y 297.329,Z 318.964,A -85,B 0,C 180,E1 -16670.766,E2 -16670.766} C_VEL
LIN {X 0,Y 298.425,Z 306.291,A -85,B 0,C 180,E1 -16671.636,E2 -16671.636} C_VEL
LIN {X 0,Y 299.265,Z 292.988,A -85,B 0,C 180,E1 -16672.248,E2 -16672.248} C_VEL
LIN {X 0,Y 299.947,Z 267.7,A -85,B 0,C 180,E1 -16672.905,E2 -16672.905} C_VEL
LIN {X 0,Y 300.74,Z 226.625,A -85,B 0,C 180,E1 -16673.897,E2 -16673.897} C_VEL
LIN {X 0,Y 294.963,Z 182.369,A -85,B 0,C 180,E1 -16675.444,E2 -16675.444} C_VEL
LIN {X 0,Y 295.391,Z 177.031,A -85,B 0,C 180,E1 -16676.875,E2 -16676.875} C_VEL
LIN {X 0,Y 293.108,Z 165.231,A -85,B 0,C 180,E1 -16680.323,E2 -16680.323} C_VEL
LIN {X 0,Y 291.411,Z 157.185,A -85,B 0,C 180,E1 -16682.82,E2 -16682.82} C_VEL
LIN {X 0,Y 291.415,Z 157.185,A -85,B 0,C 180,E1 -16687.079,E2 -16687.079} C_VEL
LIN {X 0,Y 291.335,Z 157.193,A -85,B 0,C 180,E1 -16690.642,E2 -16690.642} C_VEL
LIN {X 0,Y 291.291,Z 157.199,A -85,B 0,C 180,E1 -16694.401,E2 -16694.401} C_VEL
LIN {X 0,Y 291.327,Z 157.195,A -85,B 0,C 180,E1 -16698.404,E2 -16698.404} C_VEL
LIN {X 0,Y 291.354,Z 157.193,A -85,B 0,C 180,E1 -16701.158,E2 -16701.158} C_VEL
LIN {X 0,Y 291.361,Z 157.19,A -85,B 0,C 180,E1 -16704.626,E2 -16704.626} C_VEL
LIN {X 0,Y 291.372,Z 157.189,A -85,B 0,C 180,E1 -16707.95,E2 -16707.95} C_VEL
LIN {X 0,Y 291.386,Z 157.19,A -85,B 0,C 180,E1 -16711.158,E2 -16711.158} C_VEL
LIN {X 0,Y 291.42,Z 157.182,A -85,B 0,C 180,E1 -16714.272,E2 -16714.272} C_VEL
LIN {X 0,Y 291.372,Z 157.19,A -85,B 0,C 180,E1 -16717.298,E2 -16717.298} C_VEL
LIN {X 0,Y 291.439,Z 157.172,A -85,B 0,C 180,E1 -16720.269,E2 -16720.269} C_VEL
LIN {X 0,Y 291.497,Z 157.166,A -85,B 0,C 180,E1 -16724.665,E2 -16724.665} C_VEL
LIN {X 0,Y 291.529,Z 157.172,A -85,B 0,C 180,E1 -16728.88,E2 -16728.88} C_VEL
LIN {X 0,Y 291.653,Z 157.151,A -85,B 0,C 180,E1 -16731.687,E2 -16731.687} C_VEL
LIN {X 0,Y 291.61,Z 157.155,A -85,B 0,C 180,E1 -16734.468,E2 -16734.468} C_VEL
LIN {X 0,Y 291.888,Z 157.127,A -85,B 0,C 180,E1 -16738.62,E2 -16738.62} C_VEL
LIN {X 0,Y 291.888,Z 157.119,A -85,B 0,C 180,E1 -16741.379,E2 -16741.379} C_VEL
LIN {X 0,Y 291.735,Z 157.144,A -85,B 0,C 180,E1 -16746.918,E2 -16746.918} C_VEL
LIN {X 0,Y 291.574,Z 157.16,A -85,B 0,C 180,E1 -16749.713,E2 -16749.713} C_VEL
LIN {X 0,Y 291.521,Z 157.169,A -85,B 0,C 180,E1 -16753.95,E2 -16753.95} C_VEL
LIN {X 0,Y 291.485,Z 157.175,A -85,B 0,C 180,E1 -16756.818,E2 -16756.818} C_VEL
LIN {X 0,Y 291.45,Z 157.178,A -85,B 0,C 180,E1 -16759.875,E2 -16759.875} C_VEL
LIN {X 0,Y 291.382,Z 157.191,A -85,B 0,C 180,E1 -16764.207,E2 -16764.207} C_VEL
LIN {X 0,Y 291.42,Z 157.182,A -85,B 0,C 180,E1 -16767.272,E2 -16767.272} C_VEL
LIN {X 0,Y 291.333,Z 157.19,A -85,B 0,C 180,E1 -16770.437,E2 -16770.437} C_VEL
LIN {X 0,Y 291.343,Z 157.193,A -85,B 0,C 180,E1 -16773.698,E2 -16773.698} C_VEL
LIN {X 0,Y 291.371,Z 157.186,A -85,B 0,C 180,E1 -16777.253,E2 -16777.253} C_VEL
LIN {X 0,Y 291.331,Z 157.192,A -85,B 0,C 180,E1 -16780.643,E2 -16780.643} C_VEL
LIN {X 0,Y 291.288,Z 157.196,A -85,B 0,C 180,E1 -16784.402,E2 -16784.402} C_VEL
LIN {X 0,Y 291.325,Z 157.194,A -85,B 0,C 180,E1 -16788.404,E2 -16788.404} C_VEL
LIN {X 0,Y 291.352,Z 157.191,A -85,B 0,C 180,E1 -16791.158,E2 -16791.158} C_VEL
LIN {X 0,Y 291.36,Z 157.19,A -85,B 0,C 180,E1 -16794.626,E2 -16794.626} C_VEL
LIN {X 0,Y 291.371,Z 157.183,A -85,B 0,C 180,E1 -16797.951,E2 -16797.951} C_VEL
LIN {X 0,Y 291.384,Z 157.189,A -85,B 0,C 180,E1 -16801.159,E2 -16801.159} C_VEL
LIN {X 0,Y 291.419,Z 157.181,A -85,B 0,C 180,E1 -16804.272,E2 -16804.272} C_VEL
LIN {X 0,Y 291.371,Z 157.192,A -85,B 0,C 180,E1 -16807.299,E2 -16807.299} C_VEL
LIN {X 0,Y 291.438,Z 157.18,A -85,B 0,C 180,E1 -16810.269,E2 -16810.269} C_VEL
LIN {X 0,Y 291.497,Z 157.175,A -85,B 0,C 180,E1 -16814.665,E2 -16814.665} C_VEL
LIN {X 0,Y 291.529,Z 157.172,A -85,B 0,C 180,E1 -16818.881,E2 -16818.881} C_VEL
LIN {X 0,Y 291.652,Z 157.15,A -85,B 0,C 180,E1 -16821.687,E2 -16821.687} C_VEL
LIN {X 0,Y 291.637,Z 157.264,A -85,B 0,C 180,E1 -16824.209,E2 -16824.209} C_VEL
LIN {X 0,Y 291.75,Z 157.93,A -85,B 0,C 180,E1 -16824.428,E2 -16824.428} C_VEL
LIN {X 0,Y 300.393,Z 182.076,A -85,B 0,C 180,E1 -16825.683,E2 -16825.683} C_VEL
LIN {X 0,Y 301.564,Z 186.96,A -85,B 0,C 180,E1 -16825.887,E2 -16825.887} C_VEL
LIN {X 0,Y 299.66,Z 264.876,A -85,B 0,C 180,E1 -16827.774,E2 -16827.774} C_VEL
LIN {X 0,Y 299.053,Z 278.16,A -85,B 0,C 180,E1 -16828.359,E2 -16828.359} C_VEL
LIN {X 0,Y 298.256,Z 291.455,A -85,B 0,C 180,E1 -16829.241,E2 -16829.241} C_VEL
LIN {X 0,Y 297.173,Z 303.517,A -85,B 0,C 180,E1 -16830.339,E2 -16830.339} C_VEL
LIN {X 0,Y 296.021,Z 314.175,A -85,B 0,C 180,E1 -16831.583,E2 -16831.583} C_VEL
LIN {X 0,Y 294.811,Z 324.41,A -85,B 0,C 180,E1 -16833.075,E2 -16833.075} C_VEL
LIN {X 0,Y 293.545,Z 333.984,A -85,B 0,C 180,E1 -16834.807,E2 -16834.807} C_VEL
LIN {X 0,Y 292.301,Z 343.2,A -85,B 0,C 180,E1 -16836.905,E2 -16836.905} C_VEL
LIN {X 0,Y 291.332,Z 350.623,A -85,B 0,C 180,E1 -16839.024,E2 -16839.024} C_VEL
LIN {X 0,Y 290.598,Z 356.512,A -85,B 0,C 180,E1 -16841.156,E2 -16841.156} C_VEL
LIN {X 0,Y 290.085,Z 361.135,A -85,B 0,C 180,E1 -16843.307,E2 -16843.307} C_VEL
LIN {X 0,Y 289.653,Z 364.642,A -85,B 0,C 180,E1 -16845.48,E2 -16845.48} C_VEL
LIN {X 0,Y 289.467,Z 366.381,A -85,B 0,C 180,E1 -16846.939,E2 -16846.939} C_VEL
LIN {X 0,Y 289.394,Z 367.898,A -85,B 0,C 180,E1 -16848.716,E2 -16848.716} C_VEL
LIN {X 0,Y 289.437,Z 368.924,A -85,B 0,C 180,E1 -16851.36,E2 -16851.36} C_VEL
LIN {X 0,Y 289.575,Z 368.902,A -85,B 0,C 180,E1 -16852.85,E2 -16852.85} C_VEL
LIN {X 0,Y 289.788,Z 368.402,A -85,B 0,C 180,E1 -16854.349,E2 -16854.349} C_VEL
LIN {X 0,Y 290.252,Z 367.019,A -85,B 0,C 180,E1 -16856.377,E2 -16856.377} C_VEL
LIN {X 0,Y 291.124,Z 364.079,A -85,B 0,C 180,E1 -16858.87,E2 -16858.87} C_VEL
LIN {X 0,Y 292.147,Z 360.167,A -85,B 0,C 180,E1 -16861.146,E2 -16861.146} C_VEL
LIN {X 0,Y 293.543,Z 354.925,A -85,B 0,C 180,E1 -16863.413,E2 -16863.413} C_VEL
LIN {X 0,Y 295.135,Z 348.727,A -85,B 0,C 180,E1 -16865.498,E2 -16865.498} C_VEL
LIN {X 0,Y 297.067,Z 341.054,A -85,B 0,C 180,E1 -16867.531,E2 -16867.531} C_VEL
LIN {X 0,Y 299.019,Z 332.296,A -85,B 0,C 180,E1 -16869.39,E2 -16869.39} C_VEL
LIN {X 0,Y 300.856,Z 323.788,A -85,B 0,C 180,E1 -16870.85,E2 -16870.85} C_VEL
LIN {X 0,Y 302.854,Z 313.393,A -85,B 0,C 180,E1 -16872.297,E2 -16872.297} C_VEL
LIN {X 0,Y 304.689,Z 301.885,A -85,B 0,C 180,E1 -16873.559,E2 -16873.559} C_VEL
LIN {X 0,Y 306.123,Z 290.478,A -85,B 0,C 180,E1 -16874.525,E2 -16874.525} C_VEL
LIN {X 0,Y 307.382,Z 277.324,A -85,B 0,C 180,E1 -16875.34,E2 -16875.34} C_VEL
LIN {X 0,Y 308.189,Z 264.428,A -85,B 0,C 180,E1 -16875.859,E2 -16875.859} C_VEL
LIN {X 0,Y 310.502,Z 196.304,A -85,B 0,C 180,E1 -16877.496,E2 -16877.496} C_VEL
LIN {X 0,Y 303.663,Z 181.218,A -85,B 0,C 180,E1 -16878.781,E2 -16878.781} C_VEL
LIN {X 0,Y 295.947,Z 166.77,A -85,B 0,C 180,E1 -16880.261,E2 -16880.261} C_VEL
LIN {X 0,Y 291.925,Z 159.437,A -85,B 0,C 180,E1 -16881.106,E2 -16881.106} C_VEL
LIN {X 0,Y 291.357,Z 157.192,A -85,B 0,C 180,E1 -16882.077,E2 -16882.077} C_VEL
LIN {X 0,Y 291.357,Z 157.186,A -85,B 0,C 180,E1 -16882.474,E2 -16882.474} C_VEL
LIN {X 0,Y 290.732,Z 157.26,A -85,B 0,C 180,E1 -16883.626,E2 -16883.626} C_VEL
LIN {X 0,Y 287.845,Z 157.632,A -85,B 0,C 180,E1 -16885.502,E2 -16885.502} C_VEL
LIN {X 0,Y 285.379,Z 157.938,A -85,B 0,C 180,E1 -16887.025,E2 -16887.025} C_VEL
LIN {X 0,Y 284.343,Z 158.067,A -85,B 0,C 180,E1 -16888.207,E2 -16888.207} C_VEL
LIN {X 0,Y 284.273,Z 158.073,A -85,B 0,C 180,E1 -16888.607,E2 -16888.607} C_VEL
LIN {X 0,Y 284.26,Z 158.076,A -85,B 0,C 180,E1 -16891.982,E2 -16891.982} C_VEL
LIN {X 0,Y 284.283,Z 158.074,A -85,B 0,C 180,E1 -16895.149,E2 -16895.149} C_VEL
LIN {X 0,Y 284.296,Z 158.066,A -85,B 0,C 180,E1 -16898.235,E2 -16898.235} C_VEL
LIN {X 0,Y 284.311,Z 158.062,A -85,B 0,C 180,E1 -16901.256,E2 -16901.256} C_VEL
LIN {X 0,Y 284.421,Z 158.048,A -85,B 0,C 180,E1 -16904.513,E2 -16904.513} C_VEL
LIN {X 0,Y 284.453,Z 158.041,A -85,B 0,C 180,E1 -16908.6,E2 -16908.6} C_VEL
LIN {X 0,Y 284.61,Z 158.032,A -85,B 0,C 180,E1 -16911.48,E2 -16911.48} C_VEL
LIN {X 0,Y 284.567,Z 158.028,A -85,B 0,C 180,E1 -16914.331,E2 -16914.331} C_VEL
LIN {X 0,Y 284.837,Z 157.991,A -85,B 0,C 180,E1 -16918.586,E2 -16918.586} C_VEL
LIN {X 0,Y 284.839,Z 158,A -85,B 0,C 180,E1 -16921.414,E2 -16921.414} C_VEL
LIN {X 0,Y 284.644,Z 158.018,A -85,B 0,C 180,E1 -16927.092,E2 -16927.092} C_VEL
LIN {X 0,Y 284.516,Z 158.046,A -85,B 0,C 180,E1 -16929.957,E2 -16929.957} C_VEL
LIN {X 0,Y 284.465,Z 158.047,A -85,B 0,C 180,E1 -16934.304,E2 -16934.304} C_VEL
LIN {X 0,Y 284.384,Z 158.052,A -85,B 0,C 180,E1 -16938.74,E2 -16938.74} C_VEL
LIN {X 0,Y 284.318,Z 158.056,A -85,B 0,C 180,E1 -16941.764,E2 -16941.764} C_VEL
LIN {X 0,Y 284.311,Z 158.07,A -85,B 0,C 180,E1 -16944.849,E2 -16944.849} C_VEL
LIN {X 0,Y 284.286,Z 158.071,A -85,B 0,C 180,E1 -16948.016,E2 -16948.016} C_VEL
LIN {X 0,Y 284.287,Z 158.067,A -85,B 0,C 180,E1 -16951.276,E2 -16951.276} C_VEL
LIN {X 0,Y 284.343,Z 158.066,A -85,B 0,C 180,E1 -16955.348,E2 -16955.348} C_VEL
LIN {X 0,Y 284.3,Z 158.068,A -85,B 0,C 180,E1 -16958.171,E2 -16958.171} C_VEL
LIN {X 0,Y 284.24,Z 158.083,A -85,B 0,C 180,E1 -16962.117,E2 -16962.117} C_VEL
LIN {X 0,Y 284.257,Z 158.078,A -85,B 0,C 180,E1 -16966.189,E2 -16966.189} C_VEL
LIN {X 0,Y 284.366,Z 158.256,A -85,B 0,C 180,E1 -16970.349,E2 -16970.349} C_VEL
LIN {X 0,Y 287.145,Z 168.199,A -85,B 0,C 180,E1 -16974.327,E2 -16974.327} C_VEL
LIN {X 0,Y 289.355,Z 177.439,A -85,B 0,C 180,E1 -16977.7,E2 -16977.7} C_VEL
LIN {X 0,Y 289.994,Z 180.33,A -85,B 0,C 180,E1 -16978.705,E2 -16978.705} C_VEL
LIN {X 0,Y 296.601,Z 194.559,A -85,B 0,C 180,E1 -16980.082,E2 -16980.082} C_VEL
LIN {X 0,Y 297.742,Z 198.465,A -85,B 0,C 180,E1 -16980.354,E2 -16980.354} C_VEL
LIN {X 0,Y 301.827,Z 220.115,A -85,B 0,C 180,E1 -16981.525,E2 -16981.525} C_VEL
LIN {X 0,Y 303.347,Z 232.551,A -85,B 0,C 180,E1 -16982.074,E2 -16982.074} C_VEL
LIN {X 0,Y 301.333,Z 289.644,A -85,B 0,C 180,E1 -16983.484,E2 -16983.484} C_VEL
LIN {X 0,Y 300.201,Z 303.134,A -85,B 0,C 180,E1 -16984.056,E2 -16984.056} C_VEL
LIN {X 0,Y 298.574,Z 315.704,A -85,B 0,C 180,E1 -16984.839,E2 -16984.839} C_VEL
LIN {X 0,Y 296.634,Z 327.736,A -85,B 0,C 180,E1 -16985.877,E2 -16985.877} C_VEL
LIN {X 0,Y 294.8,Z 337.919,A -85,B 0,C 180,E1 -16987.022,E2 -16987.022} C_VEL
LIN {X 0,Y 292.483,Z 348.515,A -85,B 0,C 180,E1 -16988.504,E2 -16988.504} C_VEL
LIN {X 0,Y 290.215,Z 358.091,A -85,B 0,C 180,E1 -16990.182,E2 -16990.182} C_VEL
LIN {X 0,Y 288.258,Z 366.264,A -85,B 0,C 180,E1 -16991.964,E2 -16991.964} C_VEL
LIN {X 0,Y 286.591,Z 373.701,A -85,B 0,C 180,E1 -16993.985,E2 -16993.985} C_VEL
LIN {X 0,Y 284.706,Z 380.855,A -85,B 0,C 180,E1 -16996.437,E2 -16996.437} C_VEL
LIN {X 0,Y 283.634,Z 385.659,A -85,B 0,C 180,E1 -16998.566,E2 -16998.566} C_VEL
LIN {X 0,Y 282.936,Z 389.371,A -85,B 0,C 180,E1 -17000.708,E2 -17000.708} C_VEL
LIN {X 0,Y 282.503,Z 392.091,A -85,B 0,C 180,E1 -17002.854,E2 -17002.854} C_VEL
LIN {X 0,Y 282.367,Z 394.306,A -85,B 0,C 180,E1 -17005.718,E2 -17005.718} C_VEL
LIN {X 0,Y 282.428,Z 394.785,A -85,B 0,C 180,E1 -17007.147,E2 -17007.147} C_VEL
LIN {X 0,Y 282.431,Z 394.867,A -85,B 0,C 180,E1 -17008.574,E2 -17008.574} C_VEL
LIN {X 0,Y 282.5,Z 394.563,A -85,B 0,C 180,E1 -17010,E2 -17010} C_VEL
LIN {X 0,Y 282.456,Z 393.861,A -85,B 0,C 180,E1 -17011.426,E2 -17011.426} C_VEL
LIN {X 0,Y 282.456,Z 392.713,A -85,B 0,C 180,E1 -17012.852,E2 -17012.852} C_VEL
LIN {X 0,Y 282.44,Z 389.384,A -85,B 0,C 180,E1 -17015.539,E2 -17015.539} C_VEL
LIN {X 0,Y 282.61,Z 385.203,A -85,B 0,C 180,E1 -17017.861,E2 -17017.861} C_VEL
LIN {X 0,Y 283.077,Z 379.142,A -85,B 0,C 180,E1 -17020.369,E2 -17020.369} C_VEL
LIN {X 0,Y 283.804,Z 372.458,A -85,B 0,C 180,E1 -17022.514,E2 -17022.514} C_VEL
LIN {X 0,Y 284.868,Z 364.141,A -85,B 0,C 180,E1 -17024.648,E2 -17024.648} C_VEL
LIN {X 0,Y 285.816,Z 356.204,A -85,B 0,C 180,E1 -17026.304,E2 -17026.304} C_VEL
LIN {X 0,Y 287.222,Z 346.244,A -85,B 0,C 180,E1 -17027.994,E2 -17027.994} C_VEL
LIN {X 0,Y 288.707,Z 334.604,A -85,B 0,C 180,E1 -17029.555,E2 -17029.555} C_VEL
LIN {X 0,Y 289.983,Z 323.137,A -85,B 0,C 180,E1 -17030.759,E2 -17030.759} C_VEL
LIN {X 0,Y 291.191,Z 311.381,A -85,B 0,C 180,E1 -17031.689,E2 -17031.689} C_VEL
LIN {X 0,Y 292.229,Z 297.862,A -85,B 0,C 180,E1 -17032.444,E2 -17032.444} C_VEL
LIN {X 0,Y 292.784,Z 284.334,A -85,B 0,C 180,E1 -17032.913,E2 -17032.913} C_VEL
LIN {X 0,Y 294.022,Z 227.549,A -85,B 0,C 180,E1 -17034.309,E2 -17034.309} C_VEL
LIN {X 0,Y 288.115,Z 182.065,A -85,B 0,C 180,E1 -17035.939,E2 -17035.939} C_VEL
LIN {X 0,Y 288.459,Z 178.946,A -85,B 0,C 180,E1 -17036.79,E2 -17036.79} C_VEL
LIN {X 0,Y 286.684,Z 169.05,A -85,B 0,C 180,E1 -17039.733,E2 -17039.733} C_VEL
LIN {X 0,Y 284.344,Z 158.065,A -85,B 0,C 180,E1 -17043.204,E2 -17043.204} C_VEL
LIN {X 0,Y 284.346,Z 158.068,A -85,B 0,C 180,E1 -17046.384,E2 -17046.384} C_VEL
LIN {X 0,Y 284.307,Z 158.072,A -85,B 0,C 180,E1 -17049.994,E2 -17049.994} C_VEL
LIN {X 0,Y 284.246,Z 158.078,A -85,B 0,C 180,E1 -17054.19,E2 -17054.19} C_VEL
LIN {X 0,Y 284.272,Z 158.075,A -85,B 0,C 180,E1 -17058.124,E2 -17058.124} C_VEL
LIN {X 0,Y 284.323,Z 158.067,A -85,B 0,C 180,E1 -17062.278,E2 -17062.278} C_VEL
LIN {X 0,Y 284.309,Z 158.072,A -85,B 0,C 180,E1 -17065.35,E2 -17065.35} C_VEL
LIN {X 0,Y 284.296,Z 158.07,A -85,B 0,C 180,E1 -17068.725,E2 -17068.725} C_VEL
LIN {X 0,Y 284.4,Z 158.058,A -85,B 0,C 180,E1 -17072.825,E2 -17072.825} C_VEL
LIN {X 0,Y 284.333,Z 158.066,A -85,B 0,C 180,E1 -17076.704,E2 -17076.704} C_VEL
LIN {X 0,Y 284.376,Z 158.051,A -85,B 0,C 180,E1 -17079.904,E2 -17079.904} C_VEL
LIN {X 0,Y 284.446,Z 158.043,A -85,B 0,C 180,E1 -17084.492,E2 -17084.492} C_VEL
LIN {X 0,Y 284.482,Z 158.047,A -85,B 0,C 180,E1 -17088.601,E2 -17088.601} C_VEL
LIN {X 0,Y 284.609,Z 158.029,A -85,B 0,C 180,E1 -17091.479,E2 -17091.479} C_VEL
LIN {X 0,Y 284.579,Z 158.03,A -85,B 0,C 180,E1 -17094.331,E2 -17094.331} C_VEL
LIN {X 0,Y 284.854,Z 158.002,A -85,B 0,C 180,E1 -17098.586,E2 -17098.586} C_VEL
LIN {X 0,Y 284.854,Z 157.995,A -85,B 0,C 180,E1 -17101.413,E2 -17101.413} C_VEL
LIN {X 0,Y 284.686,Z 158.021,A -85,B 0,C 180,E1 -17107.09,E2 -17107.09} C_VEL
LIN {X 0,Y 284.518,Z 158.04,A -85,B 0,C 180,E1 -17109.957,E2 -17109.957} C_VEL
LIN {X 0,Y 284.481,Z 158.048,A -85,B 0,C 180,E1 -17114.303,E2 -17114.303} C_VEL
LIN {X 0,Y 284.422,Z 158.053,A -85,B 0,C 180,E1 -17117.248,E2 -17117.248} C_VEL
LIN {X 0,Y 284.376,Z 158.058,A -85,B 0,C 180,E1 -17120.242,E2 -17120.242} C_VEL
LIN {X 0,Y 284.337,Z 158.064,A -85,B 0,C 180,E1 -17124.846,E2 -17124.846} C_VEL
LIN {X 0,Y 284.328,Z 158.068,A -85,B 0,C 180,E1 -17128.011,E2 -17128.011} C_VEL
LIN {X 0,Y 284.293,Z 158.066,A -85,B 0,C 180,E1 -17131.274,E2 -17131.274} C_VEL
LIN {X 0,Y 284.34,Z 158.064,A -85,B 0,C 180,E1 -17135.348,E2 -17135.348} C_VEL
LIN {X 0,Y 284.307,Z 158.066,A -85,B 0,C 180,E1 -17138.169,E2 -17138.169} C_VEL
LIN {X 0,Y 284.268,Z 158.074,A -85,B 0,C 180,E1 -17142.124,E2 -17142.124} C_VEL
LIN {X 0,Y 284.254,Z 158.074,A -85,B 0,C 180,E1 -17146.189,E2 -17146.189} C_VEL
LIN {X 0,Y 284.305,Z 158.068,A -85,B 0,C 180,E1 -17150.024,E2 -17150.024} C_VEL
LIN {X 0,Y 284.331,Z 158.069,A -85,B 0,C 180,E1 -17153.614,E2 -17153.614} C_VEL
LIN {X 0,Y 284.306,Z 158.069,A -85,B 0,C 180,E1 -17157.19,E2 -17157.19} C_VEL
LIN {X 0,Y 284.358,Z 158.06,A -85,B 0,C 180,E1 -17160.376,E2 -17160.376} C_VEL
LIN {X 0,Y 284.379,Z 158.06,A -85,B 0,C 180,E1 -17163.587,E2 -17163.587} C_VEL
LIN {X 0,Y 284.332,Z 158.063,A -85,B 0,C 180,E1 -17166.704,E2 -17166.704} C_VEL
LIN {X 0,Y 284.375,Z 158.06,A -85,B 0,C 180,E1 -17169.905,E2 -17169.905} C_VEL
LIN {X 0,Y 284.447,Z 158.052,A -85,B 0,C 180,E1 -17174.492,E2 -17174.492} C_VEL
LIN {X 0,Y 284.482,Z 158.048,A -85,B 0,C 180,E1 -17178.601,E2 -17178.601} C_VEL
LIN {X 0,Y 284.609,Z 158.026,A -85,B 0,C 180,E1 -17181.48,E2 -17181.48} C_VEL
LIN {X 0,Y 284.661,Z 158.221,A -85,B 0,C 180,E1 -17183.889,E2 -17183.889} C_VEL
LIN {X 0,Y 293.349,Z 182.64,A -85,B 0,C 180,E1 -17185.206,E2 -17185.206} C_VEL
LIN {X 0,Y 294.795,Z 187.488,A -85,B 0,C 180,E1 -17185.436,E2 -17185.436} C_VEL
LIN {X 0,Y 294.668,Z 200.572,A -85,B 0,C 180,E1 -17185.769,E2 -17185.769} C_VEL
LIN {X 0,Y 292.874,Z 265.572,A -85,B 0,C 180,E1 -17187.378,E2 -17187.378} C_VEL
LIN {X 0,Y 292.237,Z 279.455,A -85,B 0,C 180,E1 -17188.019,E2 -17188.019} C_VEL
LIN {X 0,Y 291.429,Z 291.943,A -85,B 0,C 180,E1 -17188.878,E2 -17188.878} C_VEL
LIN {X 0,Y 290.308,Z 303.961,A -85,B 0,C 180,E1 -17190,E2 -17190} C_VEL
LIN {X 0,Y 289.025,Z 315.498,A -85,B 0,C 180,E1 -17191.394,E2 -17191.394} C_VEL
LIN {X 0,Y 287.743,Z 325.876,A -85,B 0,C 180,E1 -17192.975,E2 -17192.975} C_VEL
LIN {X 0,Y 286.312,Z 336.039,A -85,B 0,C 180,E1 -17194.929,E2 -17194.929} C_VEL
LIN {X 0,Y 285.132,Z 344.943,A -85,B 0,C 180,E1 -17197.079,E2 -17197.079} C_VEL
LIN {X 0,Y 284.174,Z 352.029,A -85,B 0,C 180,E1 -17199.25,E2 -17199.25} C_VEL
LIN {X 0,Y 283.421,Z 357.704,A -85,B 0,C 180,E1 -17201.442,E2 -17201.442} C_VEL
LIN {X 0,Y 282.942,Z 362.013,A -85,B 0,C 180,E1 -17203.581,E2 -17203.581} C_VEL
LIN {X 0,Y 282.497,Z 365.46,A -85,B 0,C 180,E1 -17205.882,E2 -17205.882} C_VEL
LIN {X 0,Y 282.366,Z 367.108,A -85,B 0,C 180,E1 -17207.378,E2 -17207.378} C_VEL
LIN {X 0,Y 282.317,Z 368.288,A -85,B 0,C 180,E1 -17208.92,E2 -17208.92} C_VEL
LIN {X 0,Y 282.303,Z 368.995,A -85,B 0,C 180,E1 -17210.398,E2 -17210.398} C_VEL
LIN {X 0,Y 282.497,Z 369.236,A -85,B 0,C 180,E1 -17213.003,E2 -17213.003} C_VEL
LIN {X 0,Y 282.816,Z 368.517,A -85,B 0,C 180,E1 -17214.99,E2 -17214.99} C_VEL
LIN {X 0,Y 283.282,Z 367.284,A -85,B 0,C 180,E1 -17216.731,E2 -17216.731} C_VEL
LIN {X 0,Y 284.021,Z 364.936,A -85,B 0,C 180,E1 -17218.85,E2 -17218.85} C_VEL
LIN {X 0,Y 285.098,Z 361.222,A -85,B 0,C 180,E1 -17221.177,E2 -17221.177} C_VEL
LIN {X 0,Y 286.708,Z 355.419,A -85,B 0,C 180,E1 -17223.801,E2 -17223.801} C_VEL
LIN {X 0,Y 288.277,Z 349.643,A -85,B 0,C 180,E1 -17225.811,E2 -17225.811} C_VEL
LIN {X 0,Y 290.098,Z 342.833,A -85,B 0,C 180,E1 -17227.714,E2 -17227.714} C_VEL
LIN {X 0,Y 292.222,Z 334.089,A -85,B 0,C 180,E1 -17229.682,E2 -17229.682} C_VEL
LIN {X 0,Y 294.233,Z 325.164,A -85,B 0,C 180,E1 -17231.288,E2 -17231.288} C_VEL
LIN {X 0,Y 296.519,Z 314,A -85,B 0,C 180,E1 -17232.888,E2 -17232.888} C_VEL
LIN {X 0,Y 298.509,Z 302.034,A -85,B 0,C 180,E1 -17234.226,E2 -17234.226} C_VEL
LIN {X 0,Y 300.014,Z 290.503,A -85,B 0,C 180,E1 -17235.213,E2 -17235.213} C_VEL
LIN {X 0,Y 301.311,Z 277.477,A -85,B 0,C 180,E1 -17236.029,E2 -17236.029} C_VEL
LIN {X 0,Y 302.152,Z 264.239,A -85,B 0,C 180,E1 -17236.563,E2 -17236.563} C_VEL
LIN {X 0,Y 304.507,Z 198.298,A -85,B 0,C 180,E1 -17238.178,E2 -17238.178} C_VEL
LIN {X 0,Y 297.639,Z 183.43,A -85,B 0,C 180,E1 -17239.522,E2 -17239.522} C_VEL
LIN {X 0,Y 291.199,Z 171.252,A -85,B 0,C 180,E1 -17240.808,E2 -17240.808} C_VEL
LIN {X 0,Y 284.8,Z 159.951,A -85,B 0,C 180,E1 -17242.154,E2 -17242.154} C_VEL
LIN {X 0,Y 284.33,Z 158.056,A -85,B 0,C 180,E1 -17243.043,E2 -17243.043} C_VEL
LIN {X 0,Y 284.306,Z 158.073,A -85,B 0,C 180,E1 -17247.191,E2 -17247.191} C_VEL
LIN {X 0,Y 284.273,Z 158.073,A -85,B 0,C 180,E1 -17248.607,E2 -17248.607} C_VEL
LIN {X 0,Y 283.644,Z 158.158,A -85,B 0,C 180,E1 -17249.791,E2 -17249.791} C_VEL
LIN {X 0,Y 280.8,Z 158.509,A -85,B 0,C 180,E1 -17251.718,E2 -17251.718} C_VEL
LIN {X 0,Y 278.36,Z 158.814,A -85,B 0,C 180,E1 -17253.284,E2 -17253.284} C_VEL
LIN {X 0,Y 277.304,Z 158.94,A -85,B 0,C 180,E1 -17254.497,E2 -17254.497} C_VEL
LIN {X 0,Y 277.216,Z 158.951,A -85,B 0,C 180,E1 -17254.909,E2 -17254.909} C_VEL
LIN {X 0,Y 277.26,Z 158.95,A -85,B 0,C 180,E1 -17259.215,E2 -17259.215} C_VEL
LIN {X 0,Y 277.336,Z 158.936,A -85,B 0,C 180,E1 -17263.815,E2 -17263.815} C_VEL
LIN {X 0,Y 277.402,Z 158.921,A -85,B 0,C 180,E1 -17268.307,E2 -17268.307} C_VEL
LIN {X 0,Y 277.571,Z 158.908,A -85,B 0,C 180,E1 -17271.262,E2 -17271.262} C_VEL
LIN {X 0,Y 277.538,Z 158.902,A -85,B 0,C 180,E1 -17274.187,E2 -17274.187} C_VEL
LIN {X 0,Y 277.804,Z 158.867,A -85,B 0,C 180,E1 -17278.551,E2 -17278.551} C_VEL
LIN {X 0,Y 277.806,Z 158.875,A -85,B 0,C 180,E1 -17281.45,E2 -17281.45} C_VEL
LIN {X 0,Y 277.602,Z 158.894,A -85,B 0,C 180,E1 -17287.273,E2 -17287.273} C_VEL
LIN {X 0,Y 277.459,Z 158.924,A -85,B 0,C 180,E1 -17290.213,E2 -17290.213} C_VEL
LIN {X 0,Y 277.412,Z 158.927,A -85,B 0,C 180,E1 -17294.676,E2 -17294.676} C_VEL
LIN {X 0,Y 277.331,Z 158.934,A -85,B 0,C 180,E1 -17299.235,E2 -17299.235} C_VEL
LIN {X 0,Y 277.287,Z 158.943,A -85,B 0,C 180,E1 -17303.925,E2 -17303.925} C_VEL
LIN {X 0,Y 277.272,Z 158.94,A -85,B 0,C 180,E1 -17307.483,E2 -17307.483} C_VEL
LIN {X 0,Y 277.25,Z 158.94,A -85,B 0,C 180,E1 -17310.473,E2 -17310.473} C_VEL
LIN {X 0,Y 277.249,Z 158.942,A -85,B 0,C 180,E1 -17313.896,E2 -17313.896} C_VEL
LIN {X 0,Y 277.257,Z 158.942,A -85,B 0,C 180,E1 -17317.471,E2 -17317.471} C_VEL
LIN {X 0,Y 277.186,Z 158.957,A -85,B 0,C 180,E1 -17321.241,E2 -17321.241} C_VEL
LIN {X 0,Y 277.2,Z 158.957,A -85,B 0,C 180,E1 -17325.227,E2 -17325.227} C_VEL
LIN {X 0,Y 277.248,Z 159.104,A -85,B 0,C 180,E1 -17329.311,E2 -17329.311} C_VEL
LIN {X 0,Y 279.742,Z 167.646,A -85,B 0,C 180,E1 -17332.918,E2 -17332.918} C_VEL
LIN {X 0,Y 281.983,Z 176.43,A -85,B 0,C 180,E1 -17336.322,E2 -17336.322} C_VEL
LIN {X 0,Y 282.743,Z 179.951,A -85,B 0,C 180,E1 -17337.594,E2 -17337.594} C_VEL
LIN {X 0,Y 284.888,Z 184.319,A -85,B 0,C 180,E1 -17338.07,E2 -17338.07} C_VEL
LIN {X 0,Y 291.102,Z 197.497,A -85,B 0,C 180,E1 -17339.403,E2 -17339.403} C_VEL
LIN {X 0,Y 292.049,Z 200.563,A -85,B 0,C 180,E1 -17339.632,E2 -17339.632} C_VEL
LIN {X 0,Y 295.793,Z 220.643,A -85,B 0,C 180,E1 -17340.753,E2 -17340.753} C_VEL
LIN {X 0,Y 297.424,Z 233.289,A -85,B 0,C 180,E1 -17341.343,E2 -17341.343} C_VEL
LIN {X 0,Y 295.322,Z 289.412,A -85,B 0,C 180,E1 -17342.758,E2 -17342.758} C_VEL
LIN {X 0,Y 294.146,Z 302.833,A -85,B 0,C 180,E1 -17343.337,E2 -17343.337} C_VEL
LIN {X 0,Y 292.37,Z 315.928,A -85,B 0,C 180,E1 -17344.171,E2 -17344.171} C_VEL
LIN {X 0,Y 290.5,Z 326.993,A -85,B 0,C 180,E1 -17345.143,E2 -17345.143} C_VEL
LIN {X 0,Y 288.555,Z 337.233,A -85,B 0,C 180,E1 -17346.304,E2 -17346.304} C_VEL
LIN {X 0,Y 286.186,Z 347.874,A -85,B 0,C 180,E1 -17347.816,E2 -17347.816} C_VEL
LIN {X 0,Y 283.546,Z 358.385,A -85,B 0,C 180,E1 -17349.695,E2 -17349.695} C_VEL
LIN {X 0,Y 281.41,Z 366.853,A -85,B 0,C 180,E1 -17351.628,E2 -17351.628} C_VEL
LIN {X 0,Y 279.433,Z 374.891,A -85,B 0,C 180,E1 -17353.939,E2 -17353.939} C_VEL
LIN {X 0,Y 277.8,Z 380.85,A -85,B 0,C 180,E1 -17356.093,E2 -17356.093} C_VEL
LIN {X 0,Y 276.627,Z 385.585,A -85,B 0,C 180,E1 -17358.273,E2 -17358.273} C_VEL
LIN {X 0,Y 275.909,Z 389.233,A -85,B 0,C 180,E1 -17360.469,E2 -17360.469} C_VEL
LIN {X 0,Y 275.452,Z 391.893,A -85,B 0,C 180,E1 -17362.67,E2 -17362.67} C_VEL
LIN {X 0,Y 275.26,Z 393.542,A -85,B 0,C 180,E1 -17364.724,E2 -17364.724} C_VEL
LIN {X 0,Y 275.354,Z 394.473,A -85,B 0,C 180,E1 -17367.074,E2 -17367.074} C_VEL
LIN {X 0,Y 275.351,Z 394.527,A -85,B 0,C 180,E1 -17368.537,E2 -17368.537} C_VEL
LIN {X 0,Y 275.415,Z 394.195,A -85,B 0,C 180,E1 -17370,E2 -17370} C_VEL
LIN {X 0,Y 275.376,Z 393.45,A -85,B 0,C 180,E1 -17371.462,E2 -17371.462} C_VEL
LIN {X 0,Y 275.382,Z 392.257,A -85,B 0,C 180,E1 -17372.925,E2 -17372.925} C_VEL
LIN {X 0,Y 275.368,Z 389.113,A -85,B 0,C 180,E1 -17375.513,E2 -17375.513} C_VEL
LIN {X 0,Y 275.539,Z 384.617,A -85,B 0,C 180,E1 -17378.064,E2 -17378.064} C_VEL
LIN {X 0,Y 276.042,Z 378.447,A -85,B 0,C 180,E1 -17380.637,E2 -17380.637} C_VEL
LIN {X 0,Y 276.857,Z 371.685,A -85,B 0,C 180,E1 -17382.833,E2 -17382.833} C_VEL
LIN {X 0,Y 277.968,Z 363.272,A -85,B 0,C 180,E1 -17385.02,E2 -17385.02} C_VEL
LIN {X 0,Y 279.05,Z 354.487,A -85,B 0,C 180,E1 -17386.853,E2 -17386.853} C_VEL
LIN {X 0,Y 280.587,Z 343.87,A -85,B 0,C 180,E1 -17388.624,E2 -17388.624} C_VEL
LIN {X 0,Y 281.949,Z 333.229,A -85,B 0,C 180,E1 -17390.044,E2 -17390.044} C_VEL
LIN {X 0,Y 283.35,Z 321.426,A -85,B 0,C 180,E1 -17391.269,E2 -17391.269} C_VEL
LIN {X 0,Y 284.561,Z 309.16,A -85,B 0,C 180,E1 -17392.221,E2 -17392.221} C_VEL
LIN {X 0,Y 285.592,Z 295.797,A -85,B 0,C 180,E1 -17392.947,E2 -17392.947} C_VEL
LIN {X 0,Y 286.123,Z 281.764,A -85,B 0,C 180,E1 -17393.4,E2 -17393.4} C_VEL
LIN {X 0,Y 287.293,Z 228.432,A -85,B 0,C 180,E1 -17394.744,E2 -17394.744} C_VEL
LIN {X 0,Y 281.333,Z 181.723,A -85,B 0,C 180,E1 -17396.467,E2 -17396.467} C_VEL
LIN {X 0,Y 281.197,Z 178.036,A -85,B 0,C 180,E1 -17397.54,E2 -17397.54} C_VEL
LIN {X 0,Y 278.941,Z 166.688,A -85,B 0,C 180,E1 -17401.058,E2 -17401.058} C_VEL
LIN {X 0,Y 277.304,Z 158.943,A -85,B 0,C 180,E1 -17403.597,E2 -17403.597} C_VEL
LIN {X 0,Y 277.277,Z 158.948,A -85,B 0,C 180,E1 -17407.468,E2 -17407.468} C_VEL
LIN {X 0,Y 277.211,Z 158.954,A -85,B 0,C 180,E1 -17411.236,E2 -17411.236} C_VEL
LIN {X 0,Y 277.202,Z 158.956,A -85,B 0,C 180,E1 -17415.226,E2 -17415.226} C_VEL
LIN {X 0,Y 277.223,Z 158.956,A -85,B 0,C 180,E1 -17419.512,E2 -17419.512} C_VEL
LIN {X 0,Y 277.268,Z 158.946,A -85,B 0,C 180,E1 -17422.53,E2 -17422.53} C_VEL
LIN {X 0,Y 277.248,Z 158.949,A -85,B 0,C 180,E1 -17426.104,E2 -17426.104} C_VEL
LIN {X 0,Y 277.262,Z 158.95,A -85,B 0,C 180,E1 -17429.538,E2 -17429.538} C_VEL
LIN {X 0,Y 277.361,Z 158.935,A -85,B 0,C 180,E1 -17432.864,E2 -17432.864} C_VEL
LIN {X 0,Y 277.298,Z 158.941,A -85,B 0,C 180,E1 -17436.076,E2 -17436.076} C_VEL
LIN {X 0,Y 277.317,Z 158.93,A -85,B 0,C 180,E1 -17440.764,E2 -17440.764} C_VEL
LIN {X 0,Y 277.409,Z 158.925,A -85,B 0,C 180,E1 -17445.324,E2 -17445.324} C_VEL
LIN {X 0,Y 277.457,Z 158.921,A -85,B 0,C 180,E1 -17449.787,E2 -17449.787} C_VEL
LIN {X 0,Y 277.604,Z 158.903,A -85,B 0,C 180,E1 -17452.727,E2 -17452.727} C_VEL
LIN {X 0,Y 277.82,Z 158.878,A -85,B 0,C 180,E1 -17458.55,E2 -17458.55} C_VEL
LIN {X 0,Y 277.82,Z 158.87,A -85,B 0,C 180,E1 -17461.449,E2 -17461.449} C_VEL
LIN {X 0,Y 277.64,Z 158.897,A -85,B 0,C 180,E1 -17467.271,E2 -17467.271} C_VEL
LIN {X 0,Y 277.461,Z 158.921,A -85,B 0,C 180,E1 -17470.213,E2 -17470.213} C_VEL
LIN {X 0,Y 277.434,Z 158.926,A -85,B 0,C 180,E1 -17474.674,E2 -17474.674} C_VEL
LIN {X 0,Y 277.341,Z 158.933,A -85,B 0,C 180,E1 -17479.234,E2 -17479.234} C_VEL
LIN {X 0,Y 277.291,Z 158.945,A -85,B 0,C 180,E1 -17484.158,E2 -17484.158} C_VEL
LIN {X 0,Y 277.323,Z 158.938,A -85,B 0,C 180,E1 -17487.505,E2 -17487.505} C_VEL
LIN {X 0,Y 277.271,Z 158.941,A -85,B 0,C 180,E1 -17490.481,E2 -17490.481} C_VEL
LIN {X 0,Y 277.246,Z 158.951,A -85,B 0,C 180,E1 -17493.896,E2 -17493.896} C_VEL
LIN {X 0,Y 277.264,Z 158.944,A -85,B 0,C 180,E1 -17497.47,E2 -17497.47} C_VEL
LIN {X 0,Y 277.208,Z 158.952,A -85,B 0,C 180,E1 -17501.236,E2 -17501.236} C_VEL
LIN {X 0,Y 277.199,Z 158.952,A -85,B 0,C 180,E1 -17505.226,E2 -17505.226} C_VEL
LIN {X 0,Y 277.221,Z 158.955,A -85,B 0,C 180,E1 -17509.512,E2 -17509.512} C_VEL
LIN {X 0,Y 277.266,Z 158.944,A -85,B 0,C 180,E1 -17512.531,E2 -17512.531} C_VEL
LIN {X 0,Y 277.246,Z 158.946,A -85,B 0,C 180,E1 -17516.104,E2 -17516.104} C_VEL
LIN {X 0,Y 277.26,Z 158.944,A -85,B 0,C 180,E1 -17519.539,E2 -17519.539} C_VEL
LIN {X 0,Y 277.36,Z 158.936,A -85,B 0,C 180,E1 -17522.865,E2 -17522.865} C_VEL
LIN {X 0,Y 277.297,Z 158.938,A -85,B 0,C 180,E1 -17526.077,E2 -17526.077} C_VEL
LIN {X 0,Y 277.323,Z 158.94,A -85,B 0,C 180,E1 -17530.765,E2 -17530.765} C_VEL
LIN {X 0,Y 277.409,Z 158.929,A -85,B 0,C 180,E1 -17535.325,E2 -17535.325} C_VEL
LIN {X 0,Y 277.457,Z 158.923,A -85,B 0,C 180,E1 -17539.787,E2 -17539.787} C_VEL
LIN {X 0,Y 277.627,Z 158.903,A -85,B 0,C 180,E1 -17543.331,E2 -17543.331} C_VEL
LIN {X 0,Y 286.712,Z 184.191,A -85,B 0,C 180,E1 -17544.762,E2 -17544.762} C_VEL
LIN {X 0,Y 288.264,Z 189.203,A -85,B 0,C 180,E1 -17545.012,E2 -17545.012} C_VEL
LIN {X 0,Y 286.116,Z 266.258,A -85,B 0,C 180,E1 -17546.965,E2 -17546.965} C_VEL
LIN {X 0,Y 285.448,Z 280.017,A -85,B 0,C 180,E1 -17547.619,E2 -17547.619} C_VEL
LIN {X 0,Y 284.613,Z 292.427,A -85,B 0,C 180,E1 -17548.497,E2 -17548.497} C_VEL
LIN {X 0,Y 283.468,Z 304.398,A -85,B 0,C 180,E1 -17549.645,E2 -17549.645} C_VEL
LIN {X 0,Y 282.124,Z 315.922,A -85,B 0,C 180,E1 -17551.071,E2 -17551.071} C_VEL
LIN {X 0,Y 280.897,Z 325.653,A -85,B 0,C 180,E1 -17552.582,E2 -17552.582} C_VEL
LIN {X 0,Y 279.575,Z 334.76,A -85,B 0,C 180,E1 -17554.325,E2 -17554.325} C_VEL
LIN {X 0,Y 278.284,Z 343.947,A -85,B 0,C 180,E1 -17556.526,E2 -17556.526} C_VEL
LIN {X 0,Y 277.274,Z 351.342,A -85,B 0,C 180,E1 -17558.748,E2 -17558.748} C_VEL
LIN {X 0,Y 276.466,Z 357.223,A -85,B 0,C 180,E1 -17560.991,E2 -17560.991} C_VEL
LIN {X 0,Y 275.905,Z 361.837,A -85,B 0,C 180,E1 -17563.253,E2 -17563.253} C_VEL
LIN {X 0,Y 275.445,Z 365.334,A -85,B 0,C 180,E1 -17565.54,E2 -17565.54} C_VEL
LIN {X 0,Y 275.249,Z 367.766,A -85,B 0,C 180,E1 -17567.843,E2 -17567.843} C_VEL
LIN {X 0,Y 275.203,Z 368.823,A -85,B 0,C 180,E1 -17569.39,E2 -17569.39} C_VEL
LIN {X 0,Y 275.234,Z 369.465,A -85,B 0,C 180,E1 -17570.946,E2 -17570.946} C_VEL
LIN {X 0,Y 275.46,Z 369.558,A -85,B 0,C 180,E1 -17573.294,E2 -17573.294} C_VEL
LIN {X 0,Y 275.877,Z 368.632,A -85,B 0,C 180,E1 -17575.663,E2 -17575.663} C_VEL
LIN {X 0,Y 276.35,Z 367.413,A -85,B 0,C 180,E1 -17577.243,E2 -17577.243} C_VEL
LIN {X 0,Y 277.274,Z 364.682,A -85,B 0,C 180,E1 -17579.621,E2 -17579.621} C_VEL
LIN {X 0,Y 278.443,Z 360.749,A -85,B 0,C 180,E1 -17582.009,E2 -17582.009} C_VEL
LIN {X 0,Y 280.126,Z 355.17,A -85,B 0,C 180,E1 -17584.508,E2 -17584.508} C_VEL
LIN {X 0,Y 281.998,Z 348.672,A -85,B 0,C 180,E1 -17586.737,E2 -17586.737} C_VEL
LIN {X 0,Y 283.975,Z 341.547,A -85,B 0,C 180,E1 -17588.676,E2 -17588.676} C_VEL
LIN {X 0,Y 286.342,Z 331.933,A -85,B 0,C 180,E1 -17590.773,E2 -17590.773} C_VEL
LIN {X 0,Y 288.724,Z 321.884,A -85,B 0,C 180,E1 -17592.492,E2 -17592.492} C_VEL
LIN {X 0,Y 291.026,Z 310.4,A -85,B 0,C 180,E1 -17594.034,E2 -17594.034} C_VEL
LIN {X 0,Y 292.94,Z 298.406,A -85,B 0,C 180,E1 -17595.296,E2 -17595.296} C_VEL
LIN {X 0,Y 294.371,Z 287.201,A -85,B 0,C 180,E1 -17596.183,E2 -17596.183} C_VEL
LIN {X 0,Y 295.573,Z 274.275,A -85,B 0,C 180,E1 -17596.919,E2 -17596.919} C_VEL
LIN {X 0,Y 296.327,Z 261.245,A -85,B 0,C 180,E1 -17597.388,E2 -17597.388} C_VEL
LIN {X 0,Y 298.515,Z 200.262,A -85,B 0,C 180,E1 -17598.903,E2 -17598.903} C_VEL
LIN {X 0,Y 291.639,Z 185.435,A -85,B 0,C 180,E1 -17600.304,E2 -17600.304} C_VEL
LIN {X 0,Y 284.228,Z 171.713,A -85,B 0,C 180,E1 -17601.854,E2 -17601.854} C_VEL
LIN {X 0,Y 279.386,Z 163.536,A -85,B 0,C 180,E1 -17602.919,E2 -17602.919} C_VEL
LIN {X 0,Y 277.613,Z 160.289,A -85,B 0,C 180,E1 -17603.375,E2 -17603.375} C_VEL
LIN {X 0,Y 277.275,Z 158.935,A -85,B 0,C 180,E1 -17604.043,E2 -17604.043} C_VEL
LIN {X 0,Y 277.238,Z 158.955,A -85,B 0,C 180,E1 -17607.836,E2 -17607.836} C_VEL
LIN {X 0,Y 277.217,Z 158.952,A -85,B 0,C 180,E1 -17611.205,E2 -17611.205} C_VEL
LIN {X 0,Y 277.216,Z 158.951,A -85,B 0,C 180,E1 -17614.909,E2 -17614.909} C_VEL
LIN {X 0,Y 276.538,Z 159.042,A -85,B 0,C 180,E1 -17616.122,E2 -17616.122} C_VEL
LIN {X 0,Y 273.68,Z 159.389,A -85,B 0,C 180,E1 -17618.099,E2 -17618.099} C_VEL
LIN {X 0,Y 271.275,Z 159.695,A -85,B 0,C 180,E1 -17619.706,E2 -17619.706} C_VEL
LIN {X 0,Y 270.265,Z 159.812,A -85,B 0,C 180,E1 -17620.952,E2 -17620.952} C_VEL
LIN {X 0,Y 270.193,Z 159.82,A -85,B 0,C 180,E1 -17621.373,E2 -17621.373} C_VEL
LIN {X 0,Y 270.337,Z 159.8,A -85,B 0,C 180,E1 -17624.932,E2 -17624.932} C_VEL
LIN {X 0,Y 270.384,Z 159.792,A -85,B 0,C 180,E1 -17629.517,E2 -17629.517} C_VEL
LIN {X 0,Y 270.563,Z 159.774,A -85,B 0,C 180,E1 -17632.538,E2 -17632.538} C_VEL
LIN {X 0,Y 270.769,Z 159.742,A -85,B 0,C 180,E1 -17638.513,E2 -17638.513} C_VEL
LIN {X 0,Y 270.771,Z 159.75,A -85,B 0,C 180,E1 -17641.488,E2 -17641.488} C_VEL
LIN {X 0,Y 270.564,Z 159.769,A -85,B 0,C 180,E1 -17647.463,E2 -17647.463} C_VEL
LIN {X 0,Y 270.412,Z 159.801,A -85,B 0,C 180,E1 -17650.483,E2 -17650.483} C_VEL
LIN {X 0,Y 270.379,Z 159.804,A -85,B 0,C 180,E1 -17655.066,E2 -17655.066} C_VEL
LIN {X 0,Y 270.281,Z 159.817,A -85,B 0,C 180,E1 -17659.757,E2 -17659.757} C_VEL
LIN {X 0,Y 270.227,Z 159.823,A -85,B 0,C 180,E1 -17664.59,E2 -17664.59} C_VEL
LIN {X 0,Y 270.201,Z 159.825,A -85,B 0,C 180,E1 -17667.917,E2 -17667.917} C_VEL
LIN {X 0,Y 270.176,Z 159.825,A -85,B 0,C 180,E1 -17671.35,E2 -17671.35} C_VEL
LIN {X 0,Y 270.202,Z 159.822,A -85,B 0,C 180,E1 -17674.906,E2 -17674.906} C_VEL
LIN {X 0,Y 270.2,Z 159.828,A -85,B 0,C 180,E1 -17678.71,E2 -17678.71} C_VEL
LIN {X 0,Y 270.151,Z 159.832,A -85,B 0,C 180,E1 -17683.245,E2 -17683.245} C_VEL
LIN {X 0,Y 270.174,Z 159.834,A -85,B 0,C 180,E1 -17687.442,E2 -17687.442} C_VEL
LIN {X 0,Y 270.163,Z 159.835,A -85,B 0,C 180,E1 -17688.141,E2 -17688.141} C_VEL
LIN {X 0,Y 272.771,Z 168.775,A -85,B 0,C 180,E1 -17692.105,E2 -17692.105} C_VEL
LIN {X 0,Y 275.152,Z 177.989,A -85,B 0,C 180,E1 -17695.81,E2 -17695.81} C_VEL
LIN {X 0,Y 275.571,Z 179.669,A -85,B 0,C 180,E1 -17696.394,E2 -17696.394} C_VEL
LIN {X 0,Y 284.221,Z 197.2,A -85,B 0,C 180,E1 -17698.381,E2 -17698.381} C_VEL
LIN {X 0,Y 286.462,Z 202.896,A -85,B 0,C 180,E1 -17698.897,E2 -17698.897} C_VEL
LIN {X 0,Y 290.053,Z 222.503,A -85,B 0,C 180,E1 -17700.024,E2 -17700.024} C_VEL
LIN {X 0,Y 291.553,Z 233.54,A -85,B 0,C 180,E1 -17700.568,E2 -17700.568} C_VEL
LIN {X 0,Y 289.359,Z 289.408,A -85,B 0,C 180,E1 -17702.006,E2 -17702.006} C_VEL
LIN {X 0,Y 288.065,Z 303.391,A -85,B 0,C 180,E1 -17702.63,E2 -17702.63} C_VEL
LIN {X 0,Y 286.223,Z 316.213,A -85,B 0,C 180,E1 -17703.475,E2 -17703.475} C_VEL
LIN {X 0,Y 284.129,Z 327.911,A -85,B 0,C 180,E1 -17704.546,E2 -17704.546} C_VEL
LIN {X 0,Y 282.116,Z 337.924,A -85,B 0,C 180,E1 -17705.729,E2 -17705.729} C_VEL
LIN {X 0,Y 279.644,Z 348.384,A -85,B 0,C 180,E1 -17707.269,E2 -17707.269} C_VEL
LIN {X 0,Y 277.389,Z 356.967,A -85,B 0,C 180,E1 -17708.836,E2 -17708.836} C_VEL
LIN {X 0,Y 275.212,Z 364.905,A -85,B 0,C 180,E1 -17710.611,E2 -17710.611} C_VEL
LIN {X 0,Y 273.147,Z 372.72,A -85,B 0,C 180,E1 -17712.789,E2 -17712.789} C_VEL
LIN {X 0,Y 271.437,Z 379.017,A -85,B 0,C 180,E1 -17714.994,E2 -17714.994} C_VEL
LIN {X 0,Y 269.983,Z 384.065,A -85,B 0,C 180,E1 -17717.216,E2 -17717.216} C_VEL
LIN {X 0,Y 269.094,Z 388.007,A -85,B 0,C 180,E1 -17719.466,E2 -17719.466} C_VEL
LIN {X 0,Y 268.682,Z 390.055,A -85,B 0,C 180,E1 -17720.97,E2 -17720.97} C_VEL
LIN {X 0,Y 268.222,Z 392.937,A -85,B 0,C 180,E1 -17723.984,E2 -17723.984} C_VEL
LIN {X 0,Y 268.257,Z 394.161,A -85,B 0,C 180,E1 -17726.996,E2 -17726.996} C_VEL
LIN {X 0,Y 268.274,Z 394.187,A -85,B 0,C 180,E1 -17728.499,E2 -17728.499} C_VEL
LIN {X 0,Y 268.332,Z 393.827,A -85,B 0,C 180,E1 -17730,E2 -17730} C_VEL
LIN {X 0,Y 268.297,Z 393.026,A -85,B 0,C 180,E1 -17731.501,E2 -17731.501} C_VEL
LIN {X 0,Y 268.308,Z 391.802,A -85,B 0,C 180,E1 -17733.003,E2 -17733.003} C_VEL
LIN {X 0,Y 268.269,Z 388.924,A -85,B 0,C 180,E1 -17735.428,E2 -17735.428} C_VEL
LIN {X 0,Y 268.488,Z 384.025,A -85,B 0,C 180,E1 -17738.277,E2 -17738.277} C_VEL
LIN {X 0,Y 269.026,Z 377.754,A -85,B 0,C 180,E1 -17740.917,E2 -17740.917} C_VEL
LIN {X 0,Y 269.911,Z 370.911,A -85,B 0,C 180,E1 -17743.169,E2 -17743.169} C_VEL
LIN {X 0,Y 271.089,Z 362.375,A -85,B 0,C 180,E1 -17745.41,E2 -17745.41} C_VEL
LIN {X 0,Y 272.25,Z 353.36,A -85,B 0,C 180,E1 -17747.304,E2 -17747.304} C_VEL
LIN {X 0,Y 273.766,Z 342.676,A -85,B 0,C 180,E1 -17749.105,E2 -17749.105} C_VEL
LIN {X 0,Y 275.173,Z 331.816,A -85,B 0,C 180,E1 -17750.559,E2 -17750.559} C_VEL
LIN {X 0,Y 276.71,Z 319.651,A -85,B 0,C 180,E1 -17751.805,E2 -17751.805} C_VEL
LIN {X 0,Y 277.963,Z 306.943,A -85,B 0,C 180,E1 -17752.778,E2 -17752.778} C_VEL
LIN {X 0,Y 278.87,Z 294.496,A -85,B 0,C 180,E1 -17753.435,E2 -17753.435} C_VEL
LIN {X 0,Y 279.473,Z 277.635,A -85,B 0,C 180,E1 -17753.954,E2 -17753.954} C_VEL
LIN {X 0,Y 280.614,Z 229.28,A -85,B 0,C 180,E1 -17755.199,E2 -17755.199} C_VEL
LIN {X 0,Y 274.533,Z 181.968,A -85,B 0,C 180,E1 -17756.99,E2 -17756.99} C_VEL
LIN {X 0,Y 274.451,Z 181.177,A -85,B 0,C 180,E1 -17757.092,E2 -17757.092} C_VEL
LIN {X 0,Y 273.014,Z 172.818,A -85,B 0,C 180,E1 -17759.705,E2 -17759.705} C_VEL
LIN {X 0,Y 270.244,Z 159.825,A -85,B 0,C 180,E1 -17763.97,E2 -17763.97} C_VEL
LIN {X 0,Y 270.236,Z 159.825,A -85,B 0,C 180,E1 -17766.738,E2 -17766.738} C_VEL
LIN {X 0,Y 270.175,Z 159.83,A -85,B 0,C 180,E1 -17770.565,E2 -17770.565} C_VEL
LIN {X 0,Y 270.153,Z 159.833,A -85,B 0,C 180,E1 -17774.62,E2 -17774.62} C_VEL
LIN {X 0,Y 270.17,Z 159.831,A -85,B 0,C 180,E1 -17778.971,E2 -17778.971} C_VEL
LIN {X 0,Y 270.218,Z 159.827,A -85,B 0,C 180,E1 -17783.259,E2 -17783.259} C_VEL
LIN {X 0,Y 270.203,Z 159.827,A -85,B 0,C 180,E1 -17786.892,E2 -17786.892} C_VEL
LIN {X 0,Y 270.23,Z 159.822,A -85,B 0,C 180,E1 -17790.386,E2 -17790.386} C_VEL
LIN {X 0,Y 270.264,Z 159.819,A -85,B 0,C 180,E1 -17793.763,E2 -17793.763} C_VEL
LIN {X 0,Y 270.209,Z 159.827,A -85,B 0,C 180,E1 -17797.036,E2 -17797.036} C_VEL
LIN {X 0,Y 270.257,Z 159.808,A -85,B 0,C 180,E1 -17800.241,E2 -17800.241} C_VEL
LIN {X 0,Y 270.368,Z 159.797,A -85,B 0,C 180,E1 -17804.933,E2 -17804.933} C_VEL
LIN {X 0,Y 270.41,Z 159.799,A -85,B 0,C 180,E1 -17809.517,E2 -17809.517} C_VEL
LIN {X 0,Y 270.565,Z 159.779,A -85,B 0,C 180,E1 -17812.537,E2 -17812.537} C_VEL
LIN {X 0,Y 270.786,Z 159.754,A -85,B 0,C 180,E1 -17818.512,E2 -17818.512} C_VEL
LIN {X 0,Y 270.786,Z 159.746,A -85,B 0,C 180,E1 -17821.487,E2 -17821.487} C_VEL
LIN {X 0,Y 270.598,Z 159.774,A -85,B 0,C 180,E1 -17827.461,E2 -17827.461} C_VEL
LIN {X 0,Y 270.412,Z 159.796,A -85,B 0,C 180,E1 -17830.482,E2 -17830.482} C_VEL
LIN {X 0,Y 270.402,Z 159.8,A -85,B 0,C 180,E1 -17835.064,E2 -17835.064} C_VEL
LIN {X 0,Y 270.299,Z 159.811,A -85,B 0,C 180,E1 -17839.755,E2 -17839.755} C_VEL
LIN {X 0,Y 270.237,Z 159.822,A -85,B 0,C 180,E1 -17844.589,E2 -17844.589} C_VEL
LIN {X 0,Y 270.269,Z 159.819,A -85,B 0,C 180,E1 -17847.909,E2 -17847.909} C_VEL
LIN {X 0,Y 270.183,Z 159.822,A -85,B 0,C 180,E1 -17851.348,E2 -17851.348} C_VEL
LIN {X 0,Y 270.2,Z 159.824,A -85,B 0,C 180,E1 -17854.905,E2 -17854.905} C_VEL
LIN {X 0,Y 270.196,Z 159.82,A -85,B 0,C 180,E1 -17858.71,E2 -17858.71} C_VEL
LIN {X 0,Y 270.164,Z 159.83,A -85,B 0,C 180,E1 -17863.249,E2 -17863.249} C_VEL
LIN {X 0,Y 270.17,Z 159.83,A -85,B 0,C 180,E1 -17867.442,E2 -17867.442} C_VEL
LIN {X 0,Y 270.206,Z 159.825,A -85,B 0,C 180,E1 -17871.374,E2 -17871.374} C_VEL
LIN {X 0,Y 270.201,Z 159.828,A -85,B 0,C 180,E1 -17875.095,E2 -17875.095} C_VEL
LIN {X 0,Y 270.199,Z 159.819,A -85,B 0,C 180,E1 -17879.131,E2 -17879.131} C_VEL
LIN {X 0,Y 270.264,Z 159.818,A -85,B 0,C 180,E1 -17882.146,E2 -17882.146} C_VEL
LIN {X 0,Y 270.238,Z 159.818,A -85,B 0,C 180,E1 -17885.537,E2 -17885.537} C_VEL
LIN {X 0,Y 270.26,Z 159.818,A -85,B 0,C 180,E1 -17890.242,E2 -17890.242} C_VEL
LIN {X 0,Y 270.377,Z 159.805,A -85,B 0,C 180,E1 -17894.934,E2 -17894.934} C_VEL
LIN {X 0,Y 270.409,Z 159.801,A -85,B 0,C 180,E1 -17899.518,E2 -17899.518} C_VEL
LIN {X 0,Y 270.575,Z 159.779,A -85,B 0,C 180,E1 -17902.757,E2 -17902.757} C_VEL
LIN {X 0,Y 272.323,Z 164.452,A -85,B 0,C 180,E1 -17903.064,E2 -17903.064} C_VEL
LIN {X 0,Y 280.459,Z 186.849,A -85,B 0,C 180,E1 -17904.356,E2 -17904.356} C_VEL
LIN {X 0,Y 281.592,Z 190.321,A -85,B 0,C 180,E1 -17904.54,E2 -17904.54} C_VEL
LIN {X 0,Y 279.373,Z 266.916,A -85,B 0,C 180,E1 -17906.53,E2 -17906.53} C_VEL
LIN {X 0,Y 278.673,Z 280.578,A -85,B 0,C 180,E1 -17907.2,E2 -17907.2} C_VEL
LIN {X 0,Y 277.83,Z 292.896,A -85,B 0,C 180,E1 -17908.098,E2 -17908.098} C_VEL
LIN {X 0,Y 276.624,Z 304.843,A -85,B 0,C 180,E1 -17909.272,E2 -17909.272} C_VEL
LIN {X 0,Y 275.232,Z 316.346,A -85,B 0,C 180,E1 -17910.732,E2 -17910.732} C_VEL
LIN {X 0,Y 274.001,Z 325.869,A -85,B 0,C 180,E1 -17912.248,E2 -17912.248} C_VEL
LIN {X 0,Y 272.617,Z 335.142,A -85,B 0,C 180,E1 -17914.066,E2 -17914.066} C_VEL
LIN {X 0,Y 271.271,Z 344.324,A -85,B 0,C 180,E1 -17916.322,E2 -17916.322} C_VEL
LIN {X 0,Y 270.177,Z 352.009,A -85,B 0,C 180,E1 -17918.707,E2 -17918.707} C_VEL
LIN {X 0,Y 269.273,Z 358.418,A -85,B 0,C 180,E1 -17921.289,E2 -17921.289} C_VEL
LIN {X 0,Y 268.734,Z 362.839,A -85,B 0,C 180,E1 -17923.614,E2 -17923.614} C_VEL
LIN {X 0,Y 268.421,Z 365.192,A -85,B 0,C 180,E1 -17925.179,E2 -17925.179} C_VEL
LIN {X 0,Y 268.219,Z 367.021,A -85,B 0,C 180,E1 -17926.752,E2 -17926.752} C_VEL
LIN {X 0,Y 268.113,Z 369.05,A -85,B 0,C 180,E1 -17929.325,E2 -17929.325} C_VEL
LIN {X 0,Y 268.16,Z 369.866,A -85,B 0,C 180,E1 -17931.526,E2 -17931.526} C_VEL
LIN {X 0,Y 268.404,Z 369.879,A -85,B 0,C 180,E1 -17933.587,E2 -17933.587} C_VEL
LIN {X 0,Y 268.984,Z 368.676,A -85,B 0,C 180,E1 -17936.371,E2 -17936.371} C_VEL
LIN {X 0,Y 269.509,Z 367.344,A -85,B 0,C 180,E1 -17937.995,E2 -17937.995} C_VEL
LIN {X 0,Y 270.515,Z 364.508,A -85,B 0,C 180,E1 -17940.371,E2 -17940.371} C_VEL
LIN {X 0,Y 271.899,Z 360.28,A -85,B 0,C 180,E1 -17942.875,E2 -17942.875} C_VEL
LIN {X 0,Y 273.545,Z 354.976,A -85,B 0,C 180,E1 -17945.226,E2 -17945.226} C_VEL
LIN {X 0,Y 275.771,Z 347.632,A -85,B 0,C 180,E1 -17947.708,E2 -17947.708} C_VEL
LIN {X 0,Y 277.907,Z 340.235,A -85,B 0,C 180,E1 -17949.684,E2 -17949.684} C_VEL
LIN {X 0,Y 280.289,Z 331.138,A -85,B 0,C 180,E1 -17951.641,E2 -17951.641} C_VEL
LIN {X 0,Y 282.75,Z 320.916,A -85,B 0,C 180,E1 -17953.365,E2 -17953.365} C_VEL
LIN {X 0,Y 285.015,Z 310.033,A -85,B 0,C 180,E1 -17954.823,E2 -17954.823} C_VEL
LIN {X 0,Y 286.879,Z 298.711,A -85,B 0,C 180,E1 -17956.025,E2 -17956.025} C_VEL
LIN {X 0,Y 288.469,Z 286.582,A -85,B 0,C 180,E1 -17956.987,E2 -17956.987} C_VEL
LIN {X 0,Y 289.676,Z 274.023,A -85,B 0,C 180,E1 -17957.698,E2 -17957.698} C_VEL
LIN {X 0,Y 290.395,Z 261.682,A -85,B 0,C 180,E1 -17958.146,E2 -17958.146} C_VEL
LIN {X 0,Y 292.666,Z 202.407,A -85,B 0,C 180,E1 -17959.638,E2 -17959.638} C_VEL
LIN {X 0,Y 285.656,Z 187.395,A -85,B 0,C 180,E1 -17961.126,E2 -17961.126} C_VEL
LIN {X 0,Y 277.424,Z 172.327,A -85,B 0,C 180,E1 -17962.955,E2 -17962.955} C_VEL
LIN {X 0,Y 272.156,Z 163.861,A -85,B 0,C 180,E1 -17964.173,E2 -17964.173} C_VEL
LIN {X 0,Y 270.556,Z 161.218,A -85,B 0,C 180,E1 -17964.559,E2 -17964.559} C_VEL
LIN {X 0,Y 270.308,Z 160.416,A -85,B 0,C 180,E1 -17964.797,E2 -17964.797} C_VEL
LIN {X 0,Y 270.198,Z 159.827,A -85,B 0,C 180,E1 -17965.094,E2 -17965.094} C_VEL
LIN {X 0,Y 270.171,Z 159.831,A -85,B 0,C 180,E1 -17969.142,E2 -17969.142} C_VEL
LIN {X 0,Y 270.188,Z 159.83,A -85,B 0,C 180,E1 -17972.177,E2 -17972.177} C_VEL
LIN {X 0,Y 270.182,Z 159.833,A -85,B 0,C 180,E1 -17975.564,E2 -17975.564} C_VEL
LIN {X 0,Y 270.218,Z 159.821,A -85,B 0,C 180,E1 -17980.238,E2 -17980.238} C_VEL
LIN {X 0,Y 270.193,Z 159.82,A -85,B 0,C 180,E1 -17981.373,E2 -17981.373} C_VEL
LIN {X 0,Y 269.567,Z 159.907,A -85,B 0,C 180,E1 -17982.618,E2 -17982.618} C_VEL
LIN {X 0,Y 266.779,Z 160.26,A -85,B 0,C 180,E1 -17984.647,E2 -17984.647} C_VEL
LIN {X 0,Y 264.393,Z 160.557,A -85,B 0,C 180,E1 -17986.297,E2 -17986.297} C_VEL
LIN {X 0,Y 263.366,Z 160.678,A -85,B 0,C 180,E1 -17987.575,E2 -17987.575} C_VEL
LIN {X 0,Y 263.281,Z 160.683,A -85,B 0,C 180,E1 -17988.008,E2 -17988.008} C_VEL
LIN {X 0,Y 263.473,Z 160.665,A -85,B 0,C 180,E1 -17990.791,E2 -17990.791} C_VEL
LIN {X 0,Y 263.481,Z 160.651,A -85,B 0,C 180,E1 -17993.876,E2 -17993.876} C_VEL
LIN {X 0,Y 263.733,Z 160.618,A -85,B 0,C 180,E1 -17998.473,E2 -17998.473} C_VEL
LIN {X 0,Y 263.735,Z 160.626,A -85,B 0,C 180,E1 -18001.527,E2 -18001.527} C_VEL
LIN {X 0,Y 263.528,Z 160.644,A -85,B 0,C 180,E1 -18007.663,E2 -18007.663} C_VEL
LIN {X 0,Y 263.351,Z 160.681,A -85,B 0,C 180,E1 -18010.767,E2 -18010.767} C_VEL
LIN {X 0,Y 263.326,Z 160.684,A -85,B 0,C 180,E1 -18015.48,E2 -18015.48} C_VEL
LIN {X 0,Y 263.246,Z 160.692,A -85,B 0,C 180,E1 -18020.308,E2 -18020.308} C_VEL
LIN {X 0,Y 263.17,Z 160.698,A -85,B 0,C 180,E1 -18025.296,E2 -18025.296} C_VEL
LIN {X 0,Y 263.136,Z 160.709,A -85,B 0,C 180,E1 -18028.735,E2 -18028.735} C_VEL
LIN {X 0,Y 263.13,Z 160.709,A -85,B 0,C 180,E1 -18032.289,E2 -18032.289} C_VEL
LIN {X 0,Y 263.179,Z 160.698,A -85,B 0,C 180,E1 -18036.762,E2 -18036.762} C_VEL
LIN {X 0,Y 263.093,Z 160.711,A -85,B 0,C 180,E1 -18039.875,E2 -18039.875} C_VEL
LIN {X 0,Y 263.1,Z 160.714,A -85,B 0,C 180,E1 -18043.989,E2 -18043.989} C_VEL
LIN {X 0,Y 263.138,Z 160.839,A -85,B 0,C 180,E1 -18047.005,E2 -18047.005} C_VEL
LIN {X 0,Y 265.849,Z 169.916,A -85,B 0,C 180,E1 -18051.247,E2 -18051.247} C_VEL
LIN {X 0,Y 268.251,Z 179.061,A -85,B 0,C 180,E1 -18055.067,E2 -18055.067} C_VEL
LIN {X 0,Y 270.558,Z 183.54,A -85,B 0,C 180,E1 -18055.647,E2 -18055.647} C_VEL
LIN {X 0,Y 277.907,Z 198.249,A -85,B 0,C 180,E1 -18057.415,E2 -18057.415} C_VEL
LIN {X 0,Y 280.937,Z 205.197,A -85,B 0,C 180,E1 -18058.134,E2 -18058.134} C_VEL
LIN {X 0,Y 284.656,Z 226.182,A -85,B 0,C 180,E1 -18059.367,E2 -18059.367} C_VEL
LIN {X 0,Y 285.683,Z 233.942,A -85,B 0,C 180,E1 -18059.759,E2 -18059.759} C_VEL
LIN {X 0,Y 283.529,Z 288.852,A -85,B 0,C 180,E1 -18061.206,E2 -18061.206} C_VEL
LIN {X 0,Y 282.207,Z 302.452,A -85,B 0,C 180,E1 -18061.81,E2 -18061.81} C_VEL
LIN {X 0,Y 280.307,Z 315.462,A -85,B 0,C 180,E1 -18062.668,E2 -18062.668} C_VEL
LIN {X 0,Y 278.112,Z 327.261,A -85,B 0,C 180,E1 -18063.753,E2 -18063.753} C_VEL
LIN {X 0,Y 275.964,Z 337.338,A -85,B 0,C 180,E1 -18064.951,E2 -18064.951} C_VEL
LIN {X 0,Y 273.454,Z 347.836,A -85,B 0,C 180,E1 -18066.524,E2 -18066.524} C_VEL
LIN {X 0,Y 270.789,Z 357.347,A -85,B 0,C 180,E1 -18068.294,E2 -18068.294} C_VEL
LIN {X 0,Y 268.528,Z 365.165,A -85,B 0,C 180,E1 -18070.108,E2 -18070.108} C_VEL
LIN {X 0,Y 266.362,Z 372.837,A -85,B 0,C 180,E1 -18072.336,E2 -18072.336} C_VEL
LIN {X 0,Y 264.587,Z 379.042,A -85,B 0,C 180,E1 -18074.596,E2 -18074.596} C_VEL
LIN {X 0,Y 263.048,Z 384.006,A -85,B 0,C 180,E1 -18076.873,E2 -18076.873} C_VEL
LIN {X 0,Y 262.073,Z 387.873,A -85,B 0,C 180,E1 -18079.18,E2 -18079.18} C_VEL
LIN {X 0,Y 261.317,Z 391.498,A -85,B 0,C 180,E1 -18082.272,E2 -18082.272} C_VEL
LIN {X 0,Y 261.089,Z 393.263,A -85,B 0,C 180,E1 -18084.857,E2 -18084.857} C_VEL
LIN {X 0,Y 261.163,Z 393.849,A -85,B 0,C 180,E1 -18086.915,E2 -18086.915} C_VEL
LIN {X 0,Y 261.198,Z 393.848,A -85,B 0,C 180,E1 -18088.458,E2 -18088.458} C_VEL
LIN {X 0,Y 261.252,Z 393.448,A -85,B 0,C 180,E1 -18090,E2 -18090} C_VEL
LIN {X 0,Y 261.221,Z 392.6,A -85,B 0,C 180,E1 -18091.541,E2 -18091.541} C_VEL
LIN {X 0,Y 261.213,Z 391.345,A -85,B 0,C 180,E1 -18093.084,E2 -18093.084} C_VEL
LIN {X 0,Y 261.18,Z 388.705,A -85,B 0,C 180,E1 -18095.36,E2 -18095.36} C_VEL
LIN {X 0,Y 261.311,Z 384.891,A -85,B 0,C 180,E1 -18097.728,E2 -18097.728} C_VEL
LIN {X 0,Y 261.699,Z 379.987,A -85,B 0,C 180,E1 -18100.053,E2 -18100.053} C_VEL
LIN {X 0,Y 262.386,Z 373.781,A -85,B 0,C 180,E1 -18102.373,E2 -18102.373} C_VEL
LIN {X 0,Y 263.518,Z 366.054,A -85,B 0,C 180,E1 -18104.676,E2 -18104.676} C_VEL
LIN {X 0,Y 264.621,Z 358.101,A -85,B 0,C 180,E1 -18106.589,E2 -18106.589} C_VEL
LIN {X 0,Y 265.904,Z 349.471,A -85,B 0,C 180,E1 -18108.292,E2 -18108.292} C_VEL
LIN {X 0,Y 267.46,Z 338.911,A -85,B 0,C 180,E1 -18109.974,E2 -18109.974} C_VEL
LIN {X 0,Y 268.782,Z 328.759,A -85,B 0,C 180,E1 -18111.272,E2 -18111.272} C_VEL
LIN {X 0,Y 270.215,Z 316.875,A -85,B 0,C 180,E1 -18112.458,E2 -18112.458} C_VEL
LIN {X 0,Y 271.419,Z 304.541,A -85,B 0,C 180,E1 -18113.359,E2 -18113.359} C_VEL
LIN {X 0,Y 272.306,Z 290.874,A -85,B 0,C 180,E1 -18114.035,E2 -18114.035} C_VEL
LIN {X 0,Y 273.838,Z 237.704,A -85,B 0,C 180,E1 -18115.471,E2 -18115.471} C_VEL
LIN {X 0,Y 273.924,Z 229.894,A -85,B 0,C 180,E1 -18115.684,E2 -18115.684} C_VEL
LIN {X 0,Y 268.076,Z 183.801,A -85,B 0,C 180,E1 -18117.476,E2 -18117.476} C_VEL
LIN {X 0,Y 267.319,Z 181.01,A -85,B 0,C 180,E1 -18117.655,E2 -18117.655} C_VEL
LIN {X 0,Y 265.269,Z 170.356,A -85,B 0,C 180,E1 -18121.106,E2 -18121.106} C_VEL
LIN {X 0,Y 263.206,Z 160.701,A -85,B 0,C 180,E1 -18124.441,E2 -18124.441} C_VEL
LIN {X 0,Y 263.166,Z 160.704,A -85,B 0,C 180,E1 -18127.896,E2 -18127.896} C_VEL
LIN {X 0,Y 263.124,Z 160.711,A -85,B 0,C 180,E1 -18131.893,E2 -18131.893} C_VEL
LIN {X 0,Y 263.125,Z 160.709,A -85,B 0,C 180,E1 -18136.15,E2 -18136.15} C_VEL
LIN {X 0,Y 263.106,Z 160.712,A -85,B 0,C 180,E1 -18140.127,E2 -18140.127} C_VEL
LIN {X 0,Y 263.163,Z 160.704,A -85,B 0,C 180,E1 -18144.018,E2 -18144.018} C_VEL
LIN {X 0,Y 263.133,Z 160.709,A -85,B 0,C 180,E1 -18147.711,E2 -18147.711} C_VEL
LIN {X 0,Y 263.202,Z 160.699,A -85,B 0,C 180,E1 -18151.782,E2 -18151.782} C_VEL
LIN {X 0,Y 263.202,Z 160.701,A -85,B 0,C 180,E1 -18155.212,E2 -18155.212} C_VEL
LIN {X 0,Y 263.237,Z 160.683,A -85,B 0,C 180,E1 -18159.691,E2 -18159.691} C_VEL
LIN {X 0,Y 263.31,Z 160.672,A -85,B 0,C 180,E1 -18164.519,E2 -18164.519} C_VEL
LIN {X 0,Y 263.349,Z 160.68,A -85,B 0,C 180,E1 -18169.233,E2 -18169.233} C_VEL
LIN {X 0,Y 263.528,Z 160.654,A -85,B 0,C 180,E1 -18172.337,E2 -18172.337} C_VEL
LIN {X 0,Y 263.75,Z 160.63,A -85,B 0,C 180,E1 -18178.473,E2 -18178.473} C_VEL
LIN {X 0,Y 263.751,Z 160.622,A -85,B 0,C 180,E1 -18181.527,E2 -18181.527} C_VEL
LIN {X 0,Y 263.558,Z 160.651,A -85,B 0,C 180,E1 -18187.662,E2 -18187.662} C_VEL
LIN {X 0,Y 263.355,Z 160.672,A -85,B 0,C 180,E1 -18190.766,E2 -18190.766} C_VEL
LIN {X 0,Y 263.35,Z 160.678,A -85,B 0,C 180,E1 -18195.478,E2 -18195.478} C_VEL
LIN {X 0,Y 263.262,Z 160.685,A -85,B 0,C 180,E1 -18200.306,E2 -18200.306} C_VEL
LIN {X 0,Y 263.192,Z 160.698,A -85,B 0,C 180,E1 -18205.293,E2 -18205.293} C_VEL
LIN {X 0,Y 263.165,Z 160.698,A -85,B 0,C 180,E1 -18208.731,E2 -18208.731} C_VEL
LIN {X 0,Y 263.132,Z 160.706,A -85,B 0,C 180,E1 -18212.288,E2 -18212.288} C_VEL
LIN {X 0,Y 263.189,Z 160.695,A -85,B 0,C 180,E1 -18216.765,E2 -18216.765} C_VEL
LIN {X 0,Y 263.123,Z 160.708,A -85,B 0,C 180,E1 -18221.593,E2 -18221.593} C_VEL
LIN {X 0,Y 263.121,Z 160.707,A -85,B 0,C 180,E1 -18226.016,E2 -18226.016} C_VEL
LIN {X 0,Y 263.104,Z 160.708,A -85,B 0,C 180,E1 -18230.128,E2 -18230.128} C_VEL
LIN {X 0,Y 263.162,Z 160.703,A -85,B 0,C 180,E1 -18234.018,E2 -18234.018} C_VEL
LIN {X 0,Y 263.132,Z 160.699,A -85,B 0,C 180,E1 -18237.712,E2 -18237.712} C_VEL
LIN {X 0,Y 263.201,Z 160.699,A -85,B 0,C 180,E1 -18241.783,E2 -18241.783} C_VEL
LIN {X 0,Y 263.2,Z 160.695,A -85,B 0,C 180,E1 -18245.212,E2 -18245.212} C_VEL
LIN {X 0,Y 263.237,Z 160.693,A -85,B 0,C 180,E1 -18249.692,E2 -18249.692} C_VEL
LIN {X 0,Y 263.323,Z 160.684,A -85,B 0,C 180,E1 -18254.521,E2 -18254.521} C_VEL
LIN {X 0,Y 263.349,Z 160.682,A -85,B 0,C 180,E1 -18259.234,E2 -18259.234} C_VEL
LIN {X 0,Y 263.541,Z 160.802,A -85,B 0,C 180,E1 -18262.193,E2 -18262.193} C_VEL
LIN {X 0,Y 265.452,Z 165.721,A -85,B 0,C 180,E1 -18262.51,E2 -18262.51} C_VEL
LIN {X 0,Y 273.507,Z 187.25,A -85,B 0,C 180,E1 -18263.814,E2 -18263.814} C_VEL
LIN {X 0,Y 274.98,Z 192.224,A -85,B 0,C 180,E1 -18264.072,E2 -18264.072} C_VEL
LIN {X 0,Y 272.704,Z 266.449,A -85,B 0,C 180,E1 -18266.029,E2 -18266.029} C_VEL
LIN {X 0,Y 272.028,Z 279.601,A -85,B 0,C 180,E1 -18266.668,E2 -18266.668} C_VEL
LIN {X 0,Y 271.148,Z 292.286,A -85,B 0,C 180,E1 -18267.586,E2 -18267.586} C_VEL
LIN {X 0,Y 269.992,Z 303.677,A -85,B 0,C 180,E1 -18268.695,E2 -18268.695} C_VEL
LIN {X 0,Y 268.554,Z 315.444,A -85,B 0,C 180,E1 -18270.188,E2 -18270.188} C_VEL
LIN {X 0,Y 267.194,Z 325.485,A -85,B 0,C 180,E1 -18271.792,E2 -18271.792} C_VEL
LIN {X 0,Y 265.659,Z 335.526,A -85,B 0,C 180,E1 -18273.792,E2 -18273.792} C_VEL
LIN {X 0,Y 264.44,Z 343.319,A -85,B 0,C 180,E1 -18275.72,E2 -18275.72} C_VEL
LIN {X 0,Y 263.283,Z 351.308,A -85,B 0,C 180,E1 -18278.182,E2 -18278.182} C_VEL
LIN {X 0,Y 262.318,Z 357.937,A -85,B 0,C 180,E1 -18280.81,E2 -18280.81} C_VEL
LIN {X 0,Y 261.74,Z 362.537,A -85,B 0,C 180,E1 -18283.193,E2 -18283.193} C_VEL
LIN {X 0,Y 261.255,Z 366.024,A -85,B 0,C 180,E1 -18285.606,E2 -18285.606} C_VEL
LIN {X 0,Y 261.077,Z 367.753,A -85,B 0,C 180,E1 -18287.225,E2 -18287.225} C_VEL
LIN {X 0,Y 261.044,Z 369.44,A -85,B 0,C 180,E1 -18289.56,E2 -18289.56} C_VEL
LIN {X 0,Y 261.116,Z 370.25,A -85,B 0,C 180,E1 -18292.137,E2 -18292.137} C_VEL
LIN {X 0,Y 261.38,Z 370.191,A -85,B 0,C 180,E1 -18293.909,E2 -18293.909} C_VEL
LIN {X 0,Y 261.671,Z 369.683,A -85,B 0,C 180,E1 -18295.451,E2 -18295.451} C_VEL
LIN {X 0,Y 262.397,Z 368.098,A -85,B 0,C 180,E1 -18297.888,E2 -18297.888} C_VEL
LIN {X 0,Y 263.453,Z 365.302,A -85,B 0,C 180,E1 -18300.455,E2 -18300.455} C_VEL
LIN {X 0,Y 264.837,Z 361.363,A -85,B 0,C 180,E1 -18302.957,E2 -18302.957} C_VEL
LIN {X 0,Y 266.601,Z 356.094,A -85,B 0,C 180,E1 -18305.448,E2 -18305.448} C_VEL
LIN {X 0,Y 268.823,Z 349.322,A -85,B 0,C 180,E1 -18307.893,E2 -18307.893} C_VEL
LIN {X 0,Y 271.003,Z 342.16,A -85,B 0,C 180,E1 -18309.93,E2 -18309.93} C_VEL
LIN {X 0,Y 273.441,Z 333.395,A -85,B 0,C 180,E1 -18311.933,E2 -18311.933} C_VEL
LIN {X 0,Y 275.974,Z 323.722,A -85,B 0,C 180,E1 -18313.691,E2 -18313.691} C_VEL
LIN {X 0,Y 278.391,Z 312.984,A -85,B 0,C 180,E1 -18315.237,E2 -18315.237} C_VEL
LIN {X 0,Y 280.548,Z 300.968,A -85,B 0,C 180,E1 -18316.592,E2 -18316.592} C_VEL
LIN {X 0,Y 282.233,Z 289.207,A -85,B 0,C 180,E1 -18317.603,E2 -18317.603} C_VEL
LIN {X 0,Y 283.589,Z 276.261,A -85,B 0,C 180,E1 -18318.395,E2 -18318.395} C_VEL
LIN {X 0,Y 284.512,Z 262.501,A -85,B 0,C 180,E1 -18318.922,E2 -18318.922} C_VEL
LIN {X 0,Y 286.896,Z 204.917,A -85,B 0,C 180,E1 -18320.387,E2 -18320.387} C_VEL
LIN {X 0,Y 281.569,Z 193.191,A -85,B 0,C 180,E1 -18321.576,E2 -18321.576} C_VEL
LIN {X 0,Y 274.586,Z 179.928,A -85,B 0,C 180,E1 -18323.182,E2 -18323.182} C_VEL
LIN {X 0,Y 268.29,Z 169.296,A -85,B 0,C 180,E1 -18324.691,E2 -18324.691} C_VEL
LIN {X 0,Y 266.105,Z 165.903,A -85,B 0,C 180,E1 -18325.229,E2 -18325.229} C_VEL
LIN {X 0,Y 263.757,Z 162.791,A -85,B 0,C 180,E1 -18325.802,E2 -18325.802} C_VEL
LIN {X 0,Y 263.235,Z 161.14,A -85,B 0,C 180,E1 -18326.029,E2 -18326.029} C_VEL
LIN {X 0,Y 263.17,Z 160.702,A -85,B 0,C 180,E1 -18326.349,E2 -18326.349} C_VEL
LIN {X 0,Y 263.109,Z 160.713,A -85,B 0,C 180,E1 -18329.502,E2 -18329.502} C_VEL
LIN {X 0,Y 263.113,Z 160.715,A -85,B 0,C 180,E1 -18332.994,E2 -18332.994} C_VEL
LIN {X 0,Y 263.115,Z 160.711,A -85,B 0,C 180,E1 -18336.381,E2 -18336.381} C_VEL
LIN {X 0,Y 263.207,Z 160.7,A -85,B 0,C 180,E1 -18339.689,E2 -18339.689} C_VEL
LIN {X 0,Y 263.289,Z 160.679,A -85,B 0,C 180,E1 -18344.519,E2 -18344.519} C_VEL
LIN {X 0,Y 263.281,Z 160.683,A -85,B 0,C 180,E1 -18348.008,E2 -18348.008} C_VEL
LIN {X 0,Y 262.635,Z 160.76,A -85,B 0,C 180,E1 -18349.287,E2 -18349.287} C_VEL
LIN {X 0,Y 259.869,Z 161.114,A -85,B 0,C 180,E1 -18351.375,E2 -18351.375} C_VEL
LIN {X 0,Y 256.676,Z 161.499,A -85,B 0,C 180,E1 -18353.944,E2 -18353.944} C_VEL
LIN {X 0,Y 256.321,Z 161.547,A -85,B 0,C 180,E1 -18354.831,E2 -18354.831} C_VEL
LIN {X 0,Y 256.695,Z 161.495,A -85,B 0,C 180,E1 -18358.431,E2 -18358.431} C_VEL
LIN {X 0,Y 256.697,Z 161.501,A -85,B 0,C 180,E1 -18361.569,E2 -18361.569} C_VEL
LIN {X 0,Y 256.456,Z 161.535,A -85,B 0,C 180,E1 -18366.294,E2 -18366.294} C_VEL
LIN {X 0,Y 256.429,Z 161.538,A -85,B 0,C 180,E1 -18369.465,E2 -18369.465} C_VEL
LIN {X 0,Y 256.239,Z 161.561,A -85,B 0,C 180,E1 -18374.291,E2 -18374.291} C_VEL
LIN {X 0,Y 256.183,Z 161.559,A -85,B 0,C 180,E1 -18377.564,E2 -18377.564} C_VEL
LIN {X 0,Y 256.144,Z 161.57,A -85,B 0,C 180,E1 -18381.111,E2 -18381.111} C_VEL
LIN {X 0,Y 256.135,Z 161.575,A -85,B 0,C 180,E1 -18385.112,E2 -18385.112} C_VEL
LIN {X 0,Y 256.057,Z 161.583,A -85,B 0,C 180,E1 -18389.607,E2 -18389.607} C_VEL
LIN {X 0,Y 256.068,Z 161.583,A -85,B 0,C 180,E1 -18393.293,E2 -18393.293} C_VEL
LIN {X 0,Y 256.113,Z 161.576,A -85,B 0,C 180,E1 -18397.27,E2 -18397.27} C_VEL
LIN {X 0,Y 256.06,Z 161.593,A -85,B 0,C 180,E1 -18402.178,E2 -18402.178} C_VEL
LIN {X 0,Y 256.041,Z 161.628,A -85,B 0,C 180,E1 -18405.662,E2 -18405.662} C_VEL
LIN {X 0,Y 258.449,Z 169.524,A -85,B 0,C 180,E1 -18409.589,E2 -18409.589} C_VEL
LIN {X 0,Y 260.676,Z 177.623,A -85,B 0,C 180,E1 -18413.247,E2 -18413.247} C_VEL
LIN {X 0,Y 260.982,Z 178.813,A -85,B 0,C 180,E1 -18413.659,E2 -18413.659} C_VEL
LIN {X 0,Y 263.361,Z 183.125,A -85,B 0,C 180,E1 -18414.289,E2 -18414.289} C_VEL
LIN {X 0,Y 269.163,Z 194.324,A -85,B 0,C 180,E1 -18415.777,E2 -18415.777} C_VEL
LIN {X 0,Y 274.905,Z 206.473,A -85,B 0,C 180,E1 -18417.194,E2 -18417.194} C_VEL
LIN {X 0,Y 275.848,Z 209.204,A -85,B 0,C 180,E1 -18417.443,E2 -18417.443} C_VEL
LIN {X 0,Y 279.397,Z 230.799,A -85,B 0,C 180,E1 -18418.729,E2 -18418.729} C_VEL
LIN {X 0,Y 279.934,Z 235.798,A -85,B 0,C 180,E1 -18418.972,E2 -18418.972} C_VEL
LIN {X 0,Y 277.683,Z 288.728,A -85,B 0,C 180,E1 -18420.385,E2 -18420.385} C_VEL
LIN {X 0,Y 276.367,Z 301.87,A -85,B 0,C 180,E1 -18420.976,E2 -18420.976} C_VEL
LIN {X 0,Y 274.429,Z 314.694,A -85,B 0,C 180,E1 -18421.824,E2 -18421.824} C_VEL
LIN {X 0,Y 272.142,Z 326.613,A -85,B 0,C 180,E1 -18422.924,E2 -18422.924} C_VEL
LIN {X 0,Y 269.593,Z 338.03,A -85,B 0,C 180,E1 -18424.316,E2 -18424.316} C_VEL
LIN {X 0,Y 266.988,Z 348.355,A -85,B 0,C 180,E1 -18425.92,E2 -18425.92} C_VEL
LIN {X 0,Y 264.223,Z 357.696,A -85,B 0,C 180,E1 -18427.726,E2 -18427.726} C_VEL
LIN {X 0,Y 261.854,Z 365.392,A -85,B 0,C 180,E1 -18429.579,E2 -18429.579} C_VEL
LIN {X 0,Y 259.604,Z 372.954,A -85,B 0,C 180,E1 -18431.86,E2 -18431.86} C_VEL
LIN {X 0,Y 257.752,Z 379.074,A -85,B 0,C 180,E1 -18434.177,E2 -18434.177} C_VEL
LIN {X 0,Y 256.102,Z 383.962,A -85,B 0,C 180,E1 -18436.511,E2 -18436.511} C_VEL
LIN {X 0,Y 255.071,Z 387.757,A -85,B 0,C 180,E1 -18438.879,E2 -18438.879} C_VEL
LIN {X 0,Y 254.256,Z 391.308,A -85,B 0,C 180,E1 -18442.056,E2 -18442.056} C_VEL
LIN {X 0,Y 254.015,Z 393.179,A -85,B 0,C 180,E1 -18445.239,E2 -18445.239} C_VEL
LIN {X 0,Y 254.072,Z 393.537,A -85,B 0,C 180,E1 -18446.828,E2 -18446.828} C_VEL
LIN {X 0,Y 254.122,Z 393.509,A -85,B 0,C 180,E1 -18448.415,E2 -18448.415} C_VEL
LIN {X 0,Y 254.174,Z 393.055,A -85,B 0,C 180,E1 -18450,E2 -18450} C_VEL
LIN {X 0,Y 254.146,Z 392.175,A -85,B 0,C 180,E1 -18451.584,E2 -18451.584} C_VEL
LIN {X 0,Y 254.121,Z 390.889,A -85,B 0,C 180,E1 -18453.17,E2 -18453.17} C_VEL
LIN {X 0,Y 254.087,Z 388.501,A -85,B 0,C 180,E1 -18455.277,E2 -18455.277} C_VEL
LIN {X 0,Y 254.248,Z 384.307,A -85,B 0,C 180,E1 -18457.944,E2 -18457.944} C_VEL
LIN {X 0,Y 254.675,Z 379.332,A -85,B 0,C 180,E1 -18460.333,E2 -18460.333} C_VEL
LIN {X 0,Y 255.405,Z 373.048,A -85,B 0,C 180,E1 -18462.717,E2 -18462.717} C_VEL
LIN {X 0,Y 256.41,Z 366.617,A -85,B 0,C 180,E1 -18464.686,E2 -18464.686} C_VEL
LIN {X 0,Y 257.548,Z 358.902,A -85,B 0,C 180,E1 -18466.641,E2 -18466.641} C_VEL
LIN {X 0,Y 258.738,Z 350.755,A -85,B 0,C 180,E1 -18468.345,E2 -18468.345} C_VEL
LIN {X 0,Y 260.366,Z 340.222,A -85,B 0,C 180,E1 -18470.13,E2 -18470.13} C_VEL
LIN {X 0,Y 261.919,Z 328.828,A -85,B 0,C 180,E1 -18471.651,E2 -18471.651} C_VEL
LIN {X 0,Y 263.389,Z 317.037,A -85,B 0,C 180,E1 -18472.865,E2 -18472.865} C_VEL
LIN {X 0,Y 264.7,Z 304.187,A -85,B 0,C 180,E1 -18473.833,E2 -18473.833} C_VEL
LIN {X 0,Y 265.593,Z 290.48,A -85,B 0,C 180,E1 -18474.526,E2 -18474.526} C_VEL
LIN {X 0,Y 267.256,Z 234.597,A -85,B 0,C 180,E1 -18476.065,E2 -18476.065} C_VEL
LIN {X 0,Y 267.142,Z 229.574,A -85,B 0,C 180,E1 -18476.219,E2 -18476.219} C_VEL
LIN {X 0,Y 261.537,Z 185.466,A -85,B 0,C 180,E1 -18477.988,E2 -18477.988} C_VEL
LIN {X 0,Y 260.08,Z 180.641,A -85,B 0,C 180,E1 -18478.302,E2 -18478.302} C_VEL
LIN {X 0,Y 257.708,Z 168.83,A -85,B 0,C 180,E1 -18482.284,E2 -18482.284} C_VEL
LIN {X 0,Y 256.159,Z 161.577,A -85,B 0,C 180,E1 -18484.914,E2 -18484.914} C_VEL
LIN {X 0,Y 256.089,Z 161.585,A -85,B 0,C 180,E1 -18489.138,E2 -18489.138} C_VEL
LIN {X 0,Y 256.062,Z 161.589,A -85,B 0,C 180,E1 -18493.327,E2 -18493.327} C_VEL
LIN {X 0,Y 256.072,Z 161.59,A -85,B 0,C 180,E1 -18497.818,E2 -18497.818} C_VEL
LIN {X 0,Y 256.072,Z 161.588,A -85,B 0,C 180,E1 -18500.858,E2 -18500.858} C_VEL
LIN {X 0,Y 256.109,Z 161.582,A -85,B 0,C 180,E1 -18504.811,E2 -18504.811} C_VEL
LIN {X 0,Y 256.093,Z 161.584,A -85,B 0,C 180,E1 -18508.572,E2 -18508.572} C_VEL
LIN {X 0,Y 256.143,Z 161.577,A -85,B 0,C 180,E1 -18512.196,E2 -18512.196} C_VEL
LIN {X 0,Y 256.143,Z 161.578,A -85,B 0,C 180,E1 -18515.696,E2 -18515.696} C_VEL
LIN {X 0,Y 256.149,Z 161.569,A -85,B 0,C 180,E1 -18519.103,E2 -18519.103} C_VEL
LIN {X 0,Y 256.244,Z 161.551,A -85,B 0,C 180,E1 -18524.081,E2 -18524.081} C_VEL
LIN {X 0,Y 256.29,Z 161.561,A -85,B 0,C 180,E1 -18528.933,E2 -18528.933} C_VEL
LIN {X 0,Y 256.47,Z 161.533,A -85,B 0,C 180,E1 -18532.125,E2 -18532.125} C_VEL
LIN {X 0,Y 256.495,Z 161.535,A -85,B 0,C 180,E1 -18536.858,E2 -18536.858} C_VEL
LIN {X 0,Y 256.765,Z 161.496,A -85,B 0,C 180,E1 -18540,E2 -18540} C_VEL
LIN {X 0,Y 256.498,Z 161.527,A -85,B 0,C 180,E1 -18543.141,E2 -18543.141} C_VEL
LIN {X 0,Y 256.515,Z 161.529,A -85,B 0,C 180,E1 -18547.873,E2 -18547.873} C_VEL
LIN {X 0,Y 256.294,Z 161.555,A -85,B 0,C 180,E1 -18552.672,E2 -18552.672} C_VEL
LIN {X 0,Y 256.282,Z 161.563,A -85,B 0,C 180,E1 -18556.302,E2 -18556.302} C_VEL
LIN {X 0,Y 256.152,Z 161.567,A -85,B 0,C 180,E1 -18561.117,E2 -18561.117} C_VEL
LIN {X 0,Y 256.17,Z 161.573,A -85,B 0,C 180,E1 -18565.13,E2 -18565.13} C_VEL
LIN {X 0,Y 256.103,Z 161.579,A -85,B 0,C 180,E1 -18569.601,E2 -18569.601} C_VEL
LIN {X 0,Y 256.066,Z 161.584,A -85,B 0,C 180,E1 -18573.293,E2 -18573.293} C_VEL
LIN {X 0,Y 256.118,Z 161.576,A -85,B 0,C 180,E1 -18577.272,E2 -18577.272} C_VEL
LIN {X 0,Y 256.07,Z 161.586,A -85,B 0,C 180,E1 -18582.181,E2 -18582.181} C_VEL
LIN {X 0,Y 256.06,Z 161.584,A -85,B 0,C 180,E1 -18586.673,E2 -18586.673} C_VEL
LIN {X 0,Y 256.07,Z 161.584,A -85,B 0,C 180,E1 -18590.858,E2 -18590.858} C_VEL
LIN {X 0,Y 256.129,Z 161.578,A -85,B 0,C 180,E1 -18592.868,E2 -18592.868} C_VEL
LIN {X 0,Y 256.067,Z 161.584,A -85,B 0,C 180,E1 -18596.707,E2 -18596.707} C_VEL
LIN {X 0,Y 256.113,Z 161.578,A -85,B 0,C 180,E1 -18600.401,E2 -18600.401} C_VEL
LIN {X 0,Y 256.17,Z 161.573,A -85,B 0,C 180,E1 -18604.87,E2 -18604.87} C_VEL
LIN {X 0,Y 256.148,Z 161.58,A -85,B 0,C 180,E1 -18609.104,E2 -18609.104} C_VEL
LIN {X 0,Y 256.258,Z 161.563,A -85,B 0,C 180,E1 -18614.083,E2 -18614.083} C_VEL
LIN {X 0,Y 256.29,Z 161.561,A -85,B 0,C 180,E1 -18618.933,E2 -18618.933} C_VEL
LIN {X 0,Y 256.465,Z 161.53,A -85,B 0,C 180,E1 -18621.534,E2 -18621.534} C_VEL
LIN {X 0,Y 258.111,Z 165.871,A -85,B 0,C 180,E1 -18621.849,E2 -18621.849} C_VEL
LIN {X 0,Y 262.032,Z 175.456,A -85,B 0,C 180,E1 -18622.499,E2 -18622.499} C_VEL
LIN {X 0,Y 268.199,Z 192.942,A -85,B 0,C 180,E1 -18623.546,E2 -18623.546} C_VEL
LIN {X 0,Y 265.979,Z 266.786,A -85,B 0,C 180,E1 -18625.549,E2 -18625.549} C_VEL
LIN {X 0,Y 265.278,Z 279.937,A -85,B 0,C 180,E1 -18626.203,E2 -18626.203} C_VEL
LIN {X 0,Y 264.364,Z 292.626,A -85,B 0,C 180,E1 -18627.143,E2 -18627.143} C_VEL
LIN {X 0,Y 263.177,Z 304.012,A -85,B 0,C 180,E1 -18628.279,E2 -18628.279} C_VEL
LIN {X 0,Y 261.693,Z 315.78,A -85,B 0,C 180,E1 -18629.808,E2 -18629.808} C_VEL
LIN {X 0,Y 260.218,Z 326.357,A -85,B 0,C 180,E1 -18631.548,E2 -18631.548} C_VEL
LIN {X 0,Y 258.703,Z 335.864,A -85,B 0,C 180,E1 -18633.505,E2 -18633.505} C_VEL
LIN {X 0,Y 257.269,Z 345.037,A -85,B 0,C 180,E1 -18635.88,E2 -18635.88} C_VEL
LIN {X 0,Y 256.305,Z 351.271,A -85,B 0,C 180,E1 -18637.88,E2 -18637.88} C_VEL
LIN {X 0,Y 255.375,Z 357.389,A -85,B 0,C 180,E1 -18640.305,E2 -18640.305} C_VEL
LIN {X 0,Y 254.753,Z 362.203,A -85,B 0,C 180,E1 -18642.75,E2 -18642.75} C_VEL
LIN {X 0,Y 254.335,Z 365.199,A -85,B 0,C 180,E1 -18644.728,E2 -18644.728} C_VEL
LIN {X 0,Y 253.946,Z 368.47,A -85,B 0,C 180,E1 -18647.724,E2 -18647.724} C_VEL
LIN {X 0,Y 253.945,Z 369.812,A -85,B 0,C 180,E1 -18649.787,E2 -18649.787} C_VEL
LIN {X 0,Y 254.107,Z 370.63,A -85,B 0,C 180,E1 -18652.781,E2 -18652.781} C_VEL
LIN {X 0,Y 254.375,Z 370.439,A -85,B 0,C 180,E1 -18654.484,E2 -18654.484} C_VEL
LIN {X 0,Y 254.783,Z 369.807,A -85,B 0,C 180,E1 -18656.19,E2 -18656.19} C_VEL
LIN {X 0,Y 255.47,Z 368.379,A -85,B 0,C 180,E1 -18658.319,E2 -18658.319} C_VEL
LIN {X 0,Y 256.794,Z 365.063,A -85,B 0,C 180,E1 -18661.332,E2 -18661.332} C_VEL
LIN {X 0,Y 258.346,Z 360.926,A -85,B 0,C 180,E1 -18663.896,E2 -18663.896} C_VEL
LIN {X 0,Y 260.296,Z 355.398,A -85,B 0,C 180,E1 -18666.442,E2 -18666.442} C_VEL
LIN {X 0,Y 262.406,Z 349.214,A -85,B 0,C 180,E1 -18668.655,E2 -18668.655} C_VEL
LIN {X 0,Y 265.068,Z 340.863,A -85,B 0,C 180,E1 -18671.013,E2 -18671.013} C_VEL
LIN {X 0,Y 267.703,Z 331.756,A -85,B 0,C 180,E1 -18673.046,E2 -18673.046} C_VEL
LIN {X 0,Y 270.361,Z 321.818,A -85,B 0,C 180,E1 -18674.783,E2 -18674.783} C_VEL
LIN {X 0,Y 272.643,Z 311.74,A -85,B 0,C 180,E1 -18676.201,E2 -18676.201} C_VEL
LIN {X 0,Y 274.575,Z 301.276,A -85,B 0,C 180,E1 -18677.382,E2 -18677.382} C_VEL
LIN {X 0,Y 276.285,Z 289.857,A -85,B 0,C 180,E1 -18678.381,E2 -18678.381} C_VEL
LIN {X 0,Y 277.731,Z 276.827,A -85,B 0,C 180,E1 -18679.198,E2 -18679.198} C_VEL
LIN {X 0,Y 278.676,Z 263.252,A -85,B 0,C 180,E1 -18679.734,E2 -18679.734} C_VEL
LIN {X 0,Y 281.078,Z 206.726,A -85,B 0,C 180,E1 -18681.21,E2 -18681.21} C_VEL
LIN {X 0,Y 273.82,Z 191.454,A -85,B 0,C 180,E1 -18682.918,E2 -18682.918} C_VEL
LIN {X 0,Y 266.286,Z 177.837,A -85,B 0,C 180,E1 -18684.758,E2 -18684.758} C_VEL
LIN {X 0,Y 261.17,Z 170.032,A -85,B 0,C 180,E1 -18686.053,E2 -18686.053} C_VEL
LIN {X 0,Y 259.113,Z 166.711,A -85,B 0,C 180,E1 -18686.61,E2 -18686.61} C_VEL
LIN {X 0,Y 256.849,Z 163.997,A -85,B 0,C 180,E1 -18687.203,E2 -18687.203} C_VEL
LIN {X 0,Y 256.088,Z 161.608,A -85,B 0,C 180,E1 -18687.528,E2 -18687.528} C_VEL
LIN {X 0,Y 256.078,Z 161.588,A -85,B 0,C 180,E1 -18692.189,E2 -18692.189} C_VEL
LIN {X 0,Y 256.085,Z 161.589,A -85,B 0,C 180,E1 -18695.691,E2 -18695.691} C_VEL
LIN {X 0,Y 256.122,Z 161.584,A -85,B 0,C 180,E1 -18699.101,E2 -18699.101} C_VEL
LIN {X 0,Y 256.214,Z 161.563,A -85,B 0,C 180,E1 -18704.08,E2 -18704.08} C_VEL
LIN {X 0,Y 256.272,Z 161.549,A -85,B 0,C 180,E1 -18708.933,E2 -18708.933} C_VEL
LIN {X 0,Y 256.491,Z 161.53,A -85,B 0,C 180,E1 -18712.126,E2 -18712.126} C_VEL
LIN {X 0,Y 256.321,Z 161.547,A -85,B 0,C 180,E1 -18714.831,E2 -18714.831} C_VEL
LIN {X 0,Y 255.672,Z 161.639,A -85,B 0,C 180,E1 -18716.145,E2 -18716.145} C_VEL
LIN {X 0,Y 253.098,Z 161.967,A -85,B 0,C 180,E1 -18718.297,E2 -18718.297} C_VEL
LIN {X 0,Y 250.039,Z 162.337,A -85,B 0,C 180,E1 -18720.938,E2 -18720.938} C_VEL
LIN {X 0,Y 249.607,Z 162.381,A -85,B 0,C 180,E1 -18721.848,E2 -18721.848} C_VEL
LIN {X 0,Y 249.427,Z 162.409,A -85,B 0,C 180,E1 -18726.472,E2 -18726.472} C_VEL
LIN {X 0,Y 249.345,Z 162.423,A -85,B 0,C 180,E1 -18729.737,E2 -18729.737} C_VEL
LIN {X 0,Y 249.185,Z 162.443,A -85,B 0,C 180,E1 -18734.705,E2 -18734.705} C_VEL
LIN {X 0,Y 249.118,Z 162.439,A -85,B 0,C 180,E1 -18738.079,E2 -18738.079} C_VEL
LIN {X 0,Y 249.083,Z 162.445,A -85,B 0,C 180,E1 -18741.519,E2 -18741.519} C_VEL
LIN {X 0,Y 249.087,Z 162.45,A -85,B 0,C 180,E1 -18745.46,E2 -18745.46} C_VEL
LIN {X 0,Y 249.039,Z 162.462,A -85,B 0,C 180,E1 -18748.974,E2 -18748.974} C_VEL
LIN {X 0,Y 249.029,Z 162.466,A -85,B 0,C 180,E1 -18752.426,E2 -18752.426} C_VEL
LIN {X 0,Y 249.047,Z 162.461,A -85,B 0,C 180,E1 -18756.343,E2 -18756.343} C_VEL
LIN {X 0,Y 248.986,Z 162.466,A -85,B 0,C 180,E1 -18760.482,E2 -18760.482} C_VEL
LIN {X 0,Y 249.032,Z 162.623,A -85,B 0,C 180,E1 -18764.309,E2 -18764.309} C_VEL
LIN {X 0,Y 251.247,Z 169.746,A -85,B 0,C 180,E1 -18768.092,E2 -18768.092} C_VEL
LIN {X 0,Y 253.61,Z 178.059,A -85,B 0,C 180,E1 -18772.063,E2 -18772.063} C_VEL
LIN {X 0,Y 256.004,Z 182.509,A -85,B 0,C 180,E1 -18772.763,E2 -18772.763} C_VEL
LIN {X 0,Y 260.741,Z 191.17,A -85,B 0,C 180,E1 -18774.076,E2 -18774.076} C_VEL
LIN {X 0,Y 266.437,Z 202.442,A -85,B 0,C 180,E1 -18775.572,E2 -18775.572} C_VEL
LIN {X 0,Y 270.41,Z 211.351,A -85,B 0,C 180,E1 -18776.595,E2 -18776.595} C_VEL
LIN {X 0,Y 273.809,Z 232.421,A -85,B 0,C 180,E1 -18777.891,E2 -18777.891} C_VEL
LIN {X 0,Y 274.262,Z 236.507,A -85,B 0,C 180,E1 -18778.103,E2 -18778.103} C_VEL
LIN {X 0,Y 271.932,Z 288.478,A -85,B 0,C 180,E1 -18779.518,E2 -18779.518} C_VEL
LIN {X 0,Y 270.63,Z 301.121,A -85,B 0,C 180,E1 -18780.093,E2 -18780.093} C_VEL
LIN {X 0,Y 268.629,Z 313.957,A -85,B 0,C 180,E1 -18780.945,E2 -18780.945} C_VEL
LIN {X 0,Y 266.257,Z 325.974,A -85,B 0,C 180,E1 -18782.061,E2 -18782.061} C_VEL
LIN {X 0,Y 263.515,Z 337.447,A -85,B 0,C 180,E1 -18783.466,E2 -18783.466} C_VEL
LIN {X 0,Y 260.84,Z 347.81,A -85,B 0,C 180,E1 -18785.102,E2 -18785.102} C_VEL
LIN {X 0,Y 258.262,Z 356.326,A -85,B 0,C 180,E1 -18786.76,E2 -18786.76} C_VEL
LIN {X 0,Y 255.695,Z 364.209,A -85,B 0,C 180,E1 -18788.642,E2 -18788.642} C_VEL
LIN {X 0,Y 253.261,Z 371.95,A -85,B 0,C 180,E1 -18790.97,E2 -18790.97} C_VEL
LIN {X 0,Y 250.915,Z 379.108,A -85,B 0,C 180,E1 -18793.734,E2 -18793.734} C_VEL
LIN {X 0,Y 249.176,Z 383.919,A -85,B 0,C 180,E1 -18796.128,E2 -18796.128} C_VEL
LIN {X 0,Y 248.086,Z 387.642,A -85,B 0,C 180,E1 -18798.562,E2 -18798.562} C_VEL
LIN {X 0,Y 247.573,Z 389.588,A -85,B 0,C 180,E1 -18800.193,E2 -18800.193} C_VEL
LIN {X 0,Y 247.195,Z 391.103,A -85,B 0,C 180,E1 -18801.827,E2 -18801.827} C_VEL
LIN {X 0,Y 246.923,Z 392.9,A -85,B 0,C 180,E1 -18805.101,E2 -18805.101} C_VEL
LIN {X 0,Y 246.984,Z 393.227,A -85,B 0,C 180,E1 -18806.737,E2 -18806.737} C_VEL
LIN {X 0,Y 247.048,Z 393.157,A -85,B 0,C 180,E1 -18808.37,E2 -18808.37} C_VEL
LIN {X 0,Y 247.098,Z 392.65,A -85,B 0,C 180,E1 -18810,E2 -18810} C_VEL
LIN {X 0,Y 247.073,Z 391.738,A -85,B 0,C 180,E1 -18811.63,E2 -18811.63} C_VEL
LIN {X 0,Y 247.032,Z 390.419,A -85,B 0,C 180,E1 -18813.262,E2 -18813.262} C_VEL
LIN {X 0,Y 246.99,Z 388.293,A -85,B 0,C 180,E1 -18815.178,E2 -18815.178} C_VEL
LIN {X 0,Y 247.188,Z 383.695,A -85,B 0,C 180,E1 -18818.172,E2 -18818.172} C_VEL
LIN {X 0,Y 247.667,Z 378.641,A -85,B 0,C 180,E1 -18820.629,E2 -18820.629} C_VEL
LIN {X 0,Y 248.448,Z 372.262,A -85,B 0,C 180,E1 -18823.079,E2 -18823.079} C_VEL
LIN {X 0,Y 249.647,Z 364.245,A -85,B 0,C 180,E1 -18825.512,E2 -18825.512} C_VEL
LIN {X 0,Y 250.681,Z 357.293,A -85,B 0,C 180,E1 -18827.25,E2 -18827.25} C_VEL
LIN {X 0,Y 252.386,Z 347.144,A -85,B 0,C 180,E1 -18829.309,E2 -18829.309} C_VEL
LIN {X 0,Y 253.987,Z 336.209,A -85,B 0,C 180,E1 -18831.083,E2 -18831.083} C_VEL
LIN {X 0,Y 255.508,Z 325.545,A -85,B 0,C 180,E1 -18832.435,E2 -18832.435} C_VEL
LIN {X 0,Y 257.03,Z 312.697,A -85,B 0,C 180,E1 -18833.678,E2 -18833.678} C_VEL
LIN {X 0,Y 258.299,Z 299.843,A -85,B 0,C 180,E1 -18834.568,E2 -18834.568} C_VEL
LIN {X 0,Y 259.022,Z 287.261,A -85,B 0,C 180,E1 -18835.138,E2 -18835.138} C_VEL
LIN {X 0,Y 260.587,Z 231.233,A -85,B 0,C 180,E1 -18836.699,E2 -18836.699} C_VEL
LIN {X 0,Y 255.044,Z 187.107,A -85,B 0,C 180,E1 -18838.525,E2 -18838.525} C_VEL
LIN {X 0,Y 252.803,Z 180.298,A -85,B 0,C 180,E1 -18838.984,E2 -18838.984} C_VEL
LIN {X 0,Y 250.636,Z 169.564,A -85,B 0,C 180,E1 -18842.73,E2 -18842.73} C_VEL
LIN {X 0,Y 249.11,Z 162.455,A -85,B 0,C 180,E1 -18845.386,E2 -18845.386} C_VEL
LIN {X 0,Y 249.039,Z 162.464,A -85,B 0,C 180,E1 -18848.378,E2 -18848.378} C_VEL
LIN {X 0,Y 249.01,Z 162.466,A -85,B 0,C 180,E1 -18852.792,E2 -18852.792} C_VEL
LIN {X 0,Y 249.017,Z 162.468,A -85,B 0,C 180,E1 -18857.362,E2 -18857.362} C_VEL
LIN {X 0,Y 249.044,Z 162.463,A -85,B 0,C 180,E1 -18862.2,E2 -18862.2} C_VEL
LIN {X 0,Y 249.057,Z 162.463,A -85,B 0,C 180,E1 -18865.641,E2 -18865.641} C_VEL
LIN {X 0,Y 249.053,Z 162.464,A -85,B 0,C 180,E1 -18869.473,E2 -18869.473} C_VEL
LIN {X 0,Y 249.071,Z 162.461,A -85,B 0,C 180,E1 -18873.162,E2 -18873.162} C_VEL
LIN {X 0,Y 249.061,Z 162.46,A -85,B 0,C 180,E1 -18876.73,E2 -18876.73} C_VEL
LIN {X 0,Y 249.083,Z 162.443,A -85,B 0,C 180,E1 -18880.209,E2 -18880.209} C_VEL
LIN {X 0,Y 249.196,Z 162.427,A -85,B 0,C 180,E1 -18883.618,E2 -18883.618} C_VEL
LIN {X 0,Y 249.233,Z 162.437,A -85,B 0,C 180,E1 -18888.615,E2 -18888.615} C_VEL
LIN {X 0,Y 249.419,Z 162.41,A -85,B 0,C 180,E1 -18891.9,E2 -18891.9} C_VEL
LIN {X 0,Y 249.286,Z 162.429,A -85,B 0,C 180,E1 -18895.148,E2 -18895.148} C_VEL
LIN {X 0,Y 249.675,Z 162.382,A -85,B 0,C 180,E1 -18898.387,E2 -18898.387} C_VEL
LIN {X 0,Y 249.675,Z 162.374,A -85,B 0,C 180,E1 -18901.613,E2 -18901.613} C_VEL
LIN {X 0,Y 249.441,Z 162.411,A -85,B 0,C 180,E1 -18906.712,E2 -18906.712} C_VEL
LIN {X 0,Y 249.343,Z 162.419,A -85,B 0,C 180,E1 -18909.736,E2 -18909.736} C_VEL
LIN {X 0,Y 249.205,Z 162.442,A -85,B 0,C 180,E1 -18914.703,E2 -18914.703} C_VEL
LIN {X 0,Y 249.138,Z 162.452,A -85,B 0,C 180,E1 -18918.077,E2 -18918.077} C_VEL
LIN {X 0,Y 249.083,Z 162.447,A -85,B 0,C 180,E1 -18921.518,E2 -18921.518} C_VEL
LIN {X 0,Y 249.116,Z 162.452,A -85,B 0,C 180,E1 -18925.475,E2 -18925.475} C_VEL
LIN {X 0,Y 249.072,Z 162.452,A -85,B 0,C 180,E1 -18928.989,E2 -18928.989} C_VEL
LIN {X 0,Y 249.029,Z 162.461,A -85,B 0,C 180,E1 -18932.426,E2 -18932.426} C_VEL
LIN {X 0,Y 249.052,Z 162.457,A -85,B 0,C 180,E1 -18936.341,E2 -18936.341} C_VEL
LIN {X 0,Y 249.004,Z 162.464,A -85,B 0,C 180,E1 -18940.478,E2 -18940.478} C_VEL
LIN {X 0,Y 249.001,Z 162.462,A -85,B 0,C 180,E1 -18944.879,E2 -18944.879} C_VEL
LIN {X 0,Y 249.015,Z 162.464,A -85,B 0,C 180,E1 -18947.363,E2 -18947.363} C_VEL
LIN {X 0,Y 249.043,Z 162.46,A -85,B 0,C 180,E1 -18952.2,E2 -18952.2} C_VEL
LIN {X 0,Y 249.042,Z 162.461,A -85,B 0,C 180,E1 -18955.64,E2 -18955.64} C_VEL
LIN {X 0,Y 249.051,Z 162.453,A -85,B 0,C 180,E1 -18959.473,E2 -18959.473} C_VEL
LIN {X 0,Y 249.07,Z 162.462,A -85,B 0,C 180,E1 -18963.162,E2 -18963.162} C_VEL
LIN {X 0,Y 249.06,Z 162.455,A -85,B 0,C 180,E1 -18966.731,E2 -18966.731} C_VEL
LIN {X 0,Y 249.085,Z 162.456,A -85,B 0,C 180,E1 -18970.21,E2 -18970.21} C_VEL
LIN {X 0,Y 249.195,Z 162.443,A -85,B 0,C 180,E1 -18973.619,E2 -18973.619} C_VEL
LIN {X 0,Y 249.233,Z 162.438,A -85,B 0,C 180,E1 -18978.616,E2 -18978.616} C_VEL
LIN {X 0,Y 249.42,Z 162.409,A -85,B 0,C 180,E1 -18980.895,E2 -18980.895} C_VEL
LIN {X 0,Y 250.349,Z 165.143,A -85,B 0,C 180,E1 -18981.078,E2 -18981.078} C_VEL
LIN {X 0,Y 255.344,Z 176.805,A -85,B 0,C 180,E1 -18981.927,E2 -18981.927} C_VEL
LIN {X 0,Y 261.536,Z 194.25,A -85,B 0,C 180,E1 -18983.019,E2 -18983.019} C_VEL
LIN {X 0,Y 259.278,Z 267.216,A -85,B 0,C 180,E1 -18985.049,E2 -18985.049} C_VEL
LIN {X 0,Y 258.502,Z 281.008,A -85,B 0,C 180,E1 -18985.761,E2 -18985.761} C_VEL
LIN {X 0,Y 257.522,Z 294.005,A -85,B 0,C 180,E1 -18986.774,E2 -18986.774} C_VEL
